  MoveL 9477 to (-30.25, 36.35, 135.08) mm, rotated rx 180 ry 0 rz 180 deg; joints [-35.768, -29.78, 105.46, 71.051, 38.171, -66.408]
  MoveL 9478 to (-30.25, 36.35, 135.08) mm, rotated rx 180 ry 0 rz 180 deg; joints [-35.768, -29.78, 105.46, 71.051, 38.171, -66.408]
  Call Extruder(64.93242)
  MoveL 9479 to (-30.02, 36.28, 135.08) mm, rotated rx -180 ry 0 rz -180 deg; joints [-35.728, -29.761, 105.45, 71.036, 38.13, -66.402]
  MoveL 9480 to (-30.02, 36.28, 135.08) mm, rotated rx -180 ry 0 rz -180 deg; joints [-35.728, -29.761, 105.45, 71.036, 38.13, -66.402]
  Call Extruder(65.06180)
  MoveL 9481 to (-29.8, 36.22, 135.08) mm, rotated rx -180 ry 0 rz 180 deg; joints [-35.688, -29.741, 105.44, 71.022, 38.09, -66.397]
  MoveL 9482 to (-29.8, 36.22, 135.08) mm, rotated rx -180 ry 0 rz 180 deg; joints [-35.688, -29.741, 105.44, 71.022, 38.09, -66.397]
  Call Extruder(65.18377)
  MoveL 9483 to (-29.59, 36.16, 135.08) mm, rotated rx 180 ry 0 rz 180 deg; joints [-35.651, -29.721, 105.43, 71.009, 38.053, -66.393]
  MoveL 9484 to (-29.59, 36.16, 135.08) mm, rotated rx 180 ry 0 rz 180 deg; joints [-35.651, -29.721, 105.43, 71.009, 38.053, -66.393]
  Call Extruder(65.29861)
  MoveL 9485 to (-29.38, 36.12, 135.08) mm, rotated rx -180 ry 0 rz 180 deg; joints [-35.617, -29.701, 105.42, 70.999, 38.019, -66.39]
  MoveL 9486 to (-29.38, 36.12, 135.08) mm, rotated rx -180 ry 0 rz 180 deg; joints [-35.617, -29.701, 105.42, 70.999, 38.019, -66.39]
  Call Extruder(65.41301)
  MoveL 9487 to (-29.18, 36.07, 135.08) mm, rotated rx 180 ry 0 rz 180 deg; joints [-35.584, -29.682, 105.41, 70.989, 37.986, -66.388]
  MoveL 9488 to (-29.18, 36.07, 135.08) mm, rotated rx 180 ry 0 rz 180 deg; joints [-35.584, -29.682, 105.41, 70.989, 37.986, -66.388]
  Call Extruder(65.52695)
  MoveL 9489 to (-28.97, 36.03, 135.08) mm, rotated rx 180 ry 0 rz -180 deg; joints [-35.55, -29.662, 105.4, 70.979, 37.952, -66.385]
  MoveL 9490 to (-28.97, 36.03, 135.08) mm, rotated rx 180 ry 0 rz -180 deg; joints [-35.55, -29.662, 105.4, 70.979, 37.952, -66.385]
  Call Extruder(65.64044)
  MoveL 9491 to (-28.77, 35.98, 135.08) mm, rotated rx -180 ry 0 rz 180 deg; joints [-35.517, -29.642, 105.39, 70.969, 37.918, -66.383]
  MoveL 9492 to (-28.77, 35.98, 135.08) mm, rotated rx -180 ry 0 rz 180 deg; joints [-35.517, -29.642, 105.39, 70.969, 37.918, -66.383]
  Call Extruder(65.77772)
  MoveL 9493 to (-28.52, 35.93, 135.08) mm, rotated rx -180 ry 0 rz 180 deg; joints [-35.477, -29.618, 105.377, 70.957, 37.877, -66.38]
  MoveL 9494 to (-28.52, 35.93, 135.08) mm, rotated rx -180 ry 0 rz 180 deg; joints [-35.477, -29.618, 105.377, 70.957, 37.877, -66.38]
  Call Extruder(65.91440)
  MoveL 9495 to (-28.27, 35.88, 135.08) mm, rotated rx 180 ry 0 rz 180 deg; joints [-35.437, -29.593, 105.365, 70.945, 37.837, -66.378]
  MoveL 9496 to (-28.27, 35.88, 135.08) mm, rotated rx 180 ry 0 rz 180 deg; joints [-35.437, -29.593, 105.365, 70.945, 37.837, -66.378]
  Call Extruder(66.05046)
  MoveL 9497 to (-28.02, 35.83, 135.08) mm, rotated rx 180 ry 0 rz -180 deg; joints [-35.397, -29.569, 105.352, 70.934, 37.796, -66.376]
  MoveL 9498 to (-28.02, 35.83, 135.08) mm, rotated rx 180 ry 0 rz -180 deg; joints [-35.397, -29.569, 105.352, 70.934, 37.796, -66.376]
  Call Extruder(66.18591)
  MoveL 9499 to (-27.77, 35.78, 135.08) mm, rotated rx 180 ry 0 rz 180 deg; joints [-35.357, -29.544, 105.339, 70.922, 37.756, -66.374]
  MoveL 9500 to (-27.77, 35.78, 135.08) mm, rotated rx 180 ry 0 rz 180 deg; joints [-35.357, -29.544, 105.339, 70.922, 37.756, -66.374]
  Call Extruder(66.32075)
  MoveL 9501 to (-27.52, 35.73, 135.08) mm, rotated rx -180 ry 0 rz -180 deg; joints [-35.317, -29.52, 105.327, 70.911, 37.716, -66.371]
  MoveL 9502 to (-27.52, 35.73, 135.08) mm, rotated rx -180 ry 0 rz -180 deg; joints [-35.317, -29.52, 105.327, 70.911, 37.716, -66.371]
  Call Extruder(66.45498)
  MoveL 9503 to (-27.27, 35.68, 135.08) mm, rotated rx 180 ry 0 rz 180 deg; joints [-35.277, -29.496, 105.314, 70.899, 37.675, -66.369]
  MoveL 9504 to (-27.27, 35.68, 135.08) mm, rotated rx 180 ry 0 rz 180 deg; joints [-35.277, -29.496, 105.314, 70.899, 37.675, -66.369]
  Call Extruder(66.58860)
  MoveL 9505 to (-27.03, 35.64, 135.08) mm, rotated rx 180 ry 0 rz 180 deg; joints [-35.238, -29.471, 105.302, 70.888, 37.635, -66.367]
  MoveL 9506 to (-27.03, 35.64, 135.08) mm, rotated rx 180 ry 0 rz 180 deg; joints [-35.238, -29.471, 105.302, 70.888, 37.635, -66.367]
  Call Extruder(66.75070)
  MoveL 9507 to (-26.72, 35.59, 135.08) mm, rotated rx -180 ry 0 rz 180 deg; joints [-35.191, -29.44, 105.286, 70.875, 37.587, -66.366]
  MoveL 9508 to (-26.72, 35.59, 135.08) mm, rotated rx -180 ry 0 rz 180 deg; joints [-35.191, -29.44, 105.286, 70.875, 37.587, -66.366]
  Call Extruder(66.91207)
  MoveL 9509 to (-26.41, 35.54, 135.08) mm, rotated rx -180 ry 0 rz 180 deg; joints [-35.145, -29.409, 105.269, 70.864, 37.54, -66.365]
  MoveL 9510 to (-26.41, 35.54, 135.08) mm, rotated rx -180 ry 0 rz 180 deg; joints [-35.145, -29.409, 105.269, 70.864, 37.54, -66.365]
  Call Extruder(67.07271)
  MoveL 9511 to (-26.11, 35.49, 135.08) mm, rotated rx 180 ry 0 rz 180 deg; joints [-35.098, -29.377, 105.253, 70.852, 37.493, -66.364]
  MoveL 9512 to (-26.11, 35.49, 135.08) mm, rotated rx 180 ry 0 rz 180 deg; joints [-35.098, -29.377, 105.253, 70.852, 37.493, -66.364]
  Call Extruder(67.23263)
  MoveL 9513 to (-25.8, 35.44, 135.08) mm, rotated rx 180 ry 0 rz 180 deg; joints [-35.052, -29.346, 105.237, 70.84, 37.445, -66.364]
  MoveL 9514 to (-25.8, 35.44, 135.08) mm, rotated rx 180 ry 0 rz 180 deg; joints [-35.052, -29.346, 105.237, 70.84, 37.445, -66.364]
  Call Extruder(67.39181)
  MoveL 9515 to (-25.5, 35.39, 135.08) mm, rotated rx -180 ry 0 rz 180 deg; joints [-35.006, -29.315, 105.221, 70.828, 37.398, -66.363]
  MoveL 9516 to (-25.5, 35.39, 135.08) mm, rotated rx -180 ry 0 rz 180 deg; joints [-35.006, -29.315, 105.221, 70.828, 37.398, -66.363]
  Call Extruder(67.55027)
  MoveL 9517 to (-25.19, 35.34, 135.08) mm, rotated rx 180 ry 0 rz 180 deg; joints [-34.96, -29.284, 105.205, 70.816, 37.351, -66.362]
  MoveL 9518 to (-25.19, 35.34, 135.08) mm, rotated rx 180 ry 0 rz 180 deg; joints [-34.96, -29.284, 105.205, 70.816, 37.351, -66.362]
  Call Extruder(67.74915)
  MoveL 9519 to (-24.8, 35.3, 135.08) mm, rotated rx 180 ry 0 rz 180 deg; joints [-34.904, -29.243, 105.184, 70.804, 37.294, -66.364]
  MoveL 9520 to (-24.8, 35.3, 135.08) mm, rotated rx 180 ry 0 rz 180 deg; joints [-34.904, -29.243, 105.184, 70.804, 37.294, -66.364]
  Call Extruder(67.94716)
  MoveL 9521 to (-24.42, 35.25, 135.08) mm, rotated rx -180 ry 0 rz 180 deg; joints [-34.849, -29.202, 105.162, 70.791, 37.236, -66.365]
  MoveL 9522 to (-24.42, 35.25, 135.08) mm, rotated rx -180 ry 0 rz 180 deg; joints [-34.849, -29.202, 105.162, 70.791, 37.236, -66.365]
  Call Extruder(68.14430)
  MoveL 9523 to (-24.03, 35.21, 135.08) mm, rotated rx 180 ry 0 rz 180 deg; joints [-34.794, -29.161, 105.141, 70.779, 37.179, -66.367]
  MoveL 9524 to (-24.03, 35.21, 135.08) mm, rotated rx 180 ry 0 rz 180 deg; joints [-34.794, -29.161, 105.141, 70.779, 37.179, -66.367]
  Call Extruder(68.34057)
  MoveL 9525 to (-23.64, 35.16, 135.08) mm, rotated rx -180 ry 0 rz 180 deg; joints [-34.738, -29.12, 105.119, 70.767, 37.122, -66.368]
  MoveL 9526 to (-23.64, 35.16, 135.08) mm, rotated rx -180 ry 0 rz 180 deg; joints [-34.738, -29.12, 105.119, 70.767, 37.122, -66.368]
  Call Extruder(68.58626)
  MoveL 9527 to (-23.15, 35.11, 135.08) mm, rotated rx -180 ry 0 rz 180 deg; joints [-34.671, -29.067, 105.092, 70.754, 37.052, -66.372]
  MoveL 9528 to (-23.15, 35.11, 135.08) mm, rotated rx -180 ry 0 rz 180 deg; joints [-34.671, -29.067, 105.092, 70.754, 37.052, -66.372]
  Call Extruder(68.88099)
  MoveL 9529 to (-22.56, 35.07, 135.08) mm, rotated rx 180 ry 0 rz 180 deg; joints [-34.592, -29.002, 105.058, 70.739, 36.969, -66.378]
  MoveL 9530 to (-22.56, 35.07, 135.08) mm, rotated rx 180 ry 0 rz 180 deg; joints [-34.592, -29.002, 105.058, 70.739, 36.969, -66.378]
  Call Extruder(69.17439)
  MoveL 9531 to (-21.97, 35.02, 135.08) mm, rotated rx 180 ry 0 rz 180 deg; joints [-34.512, -28.938, 105.024, 70.725, 36.886, -66.384]
  MoveL 9532 to (-21.97, 35.02, 135.08) mm, rotated rx 180 ry 0 rz 180 deg; joints [-34.512, -28.938, 105.024, 70.725, 36.886, -66.384]
  Call Extruder(69.60772)
  MoveL 9533 to (-21.1, 34.97, 135.08) mm, rotated rx 180 ry 0 rz 180 deg; joints [-34.399, -28.84, 104.973, 70.708, 36.767, -66.397]
  MoveL 9534 to (-21.1, 34.97, 135.08) mm, rotated rx 180 ry 0 rz 180 deg; joints [-34.399, -28.84, 104.973, 70.708, 36.767, -66.397]
  Call Extruder(70.17988)
  MoveL 9535 to (-19.94, 34.93, 135.08) mm, rotated rx 180 ry 0 rz 180 deg; joints [-34.253, -28.708, 104.904, 70.689, 36.613, -66.416]
  MoveL 9536 to (-19.94, 34.93, 135.08) mm, rotated rx 180 ry 0 rz 180 deg; joints [-34.253, -28.708, 104.904, 70.689, 36.613, -66.416]
  Call Extruder(70.60771)
  MoveL 9537 to (-19.06, 34.91, 135.08) mm, rotated rx 180 ry 0 rz 180 deg; joints [-34.146, -28.608, 104.85, 70.677, 36.499, -66.434]
  Call Extruder(187.25639)
  MoveL 9538 to (219.06, 34.91, 135.08) mm, rotated rx -180 ry 0 rz 180 deg; joints [-18.248, 3.511, 79.317, 69.262, 19.562, -68.108]
  MoveL 9539 to (219.06, 34.91, 135.08) mm, rotated rx -180 ry 0 rz 180 deg; joints [-18.248, 3.511, 79.317, 69.262, 19.562, -68.108]
  Call Extruder(187.97196)
  MoveL 9540 to (220.52, 34.95, 135.08) mm, rotated rx 180 ry 0 rz 180 deg; joints [-18.199, 3.735, 79.08, 69.172, 19.522, -68.02]
  MoveL 9541 to (220.52, 34.95, 135.08) mm, rotated rx 180 ry 0 rz 180 deg; joints [-18.199, 3.735, 79.08, 69.172, 19.522, -68.02]
  Call Extruder(188.54670)
  MoveL 9542 to (221.68, 35, 135.08) mm, rotated rx 180 ry 0 rz 180 deg; joints [-18.162, 3.916, 78.888, 69.101, 19.491, -67.949]
  MoveL 9543 to (221.68, 35, 135.08) mm, rotated rx 180 ry 0 rz 180 deg; joints [-18.162, 3.916, 78.888, 69.101, 19.491, -67.949]
  Call Extruder(188.84009)
  MoveL 9544 to (222.27, 35.04, 135.08) mm, rotated rx -180 ry 0 rz 180 deg; joints [-18.146, 4.008, 78.789, 69.066, 19.478, -67.915]
  MoveL 9545 to (222.27, 35.04, 135.08) mm, rotated rx -180 ry 0 rz 180 deg; joints [-18.146, 4.008, 78.789, 69.066, 19.478, -67.915]
  Call Extruder(189.13482)
  MoveL 9546 to (222.86, 35.09, 135.08) mm, rotated rx -180 ry 0 rz -180 deg; joints [-18.13, 4.101, 78.691, 69.032, 19.465, -67.88]
  MoveL 9547 to (222.86, 35.09, 135.08) mm, rotated rx -180 ry 0 rz -180 deg; joints [-18.13, 4.101, 78.691, 69.032, 19.465, -67.88]
  Call Extruder(189.43087)
  MoveL 9548 to (223.45, 35.14, 135.08) mm, rotated rx 180 ry 0 rz 180 deg; joints [-18.113, 4.194, 78.591, 68.997, 19.452, -67.846]
  MoveL 9549 to (223.45, 35.14, 135.08) mm, rotated rx 180 ry 0 rz 180 deg; joints [-18.113, 4.194, 78.591, 68.997, 19.452, -67.846]
  Call Extruder(189.62715)
  MoveL 9550 to (223.84, 35.18, 135.08) mm, rotated rx -180 ry 0 rz 180 deg; joints [-18.104, 4.256, 78.525, 68.976, 19.446, -67.824]
  MoveL 9551 to (223.84, 35.18, 135.08) mm, rotated rx -180 ry 0 rz 180 deg; joints [-18.104, 4.256, 78.525, 68.976, 19.446, -67.824]
  Call Extruder(189.82429)
  MoveL 9552 to (224.22, 35.23, 135.08) mm, rotated rx 180 ry 0 rz 180 deg; joints [-18.095, 4.318, 78.459, 68.954, 19.439, -67.802]
  MoveL 9553 to (224.22, 35.23, 135.08) mm, rotated rx 180 ry 0 rz 180 deg; joints [-18.095, 4.318, 78.459, 68.954, 19.439, -67.802]
  Call Extruder(190.02230)
  MoveL 9554 to (224.61, 35.27, 135.08) mm, rotated rx -180 ry 0 rz 180 deg; joints [-18.087, 4.38, 78.393, 68.932, 19.432, -67.78]
  MoveL 9555 to (224.61, 35.27, 135.08) mm, rotated rx -180 ry 0 rz 180 deg; joints [-18.087, 4.38, 78.393, 68.932, 19.432, -67.78]
  Call Extruder(190.22117)
  MoveL 9556 to (225, 35.32, 135.08) mm, rotated rx 180 ry 0 rz -180 deg; joints [-18.078, 4.442, 78.326, 68.91, 19.426, -67.758]
  MoveL 9557 to (225, 35.32, 135.08) mm, rotated rx 180 ry 0 rz -180 deg; joints [-18.078, 4.442, 78.326, 68.91, 19.426, -67.758]
  Call Extruder(190.40025)
  MoveL 9558 to (225.34, 35.37, 135.08) mm, rotated rx 180 ry 0 rz 180 deg; joints [-18.07, 4.497, 78.267, 68.891, 19.42, -67.739]
  MoveL 9559 to (225.34, 35.37, 135.08) mm, rotated rx 180 ry 0 rz 180 deg; joints [-18.07, 4.497, 78.267, 68.891, 19.42, -67.739]
  Call Extruder(190.55944)
  MoveL 9560 to (225.65, 35.42, 135.08) mm, rotated rx 180 ry 0 rz 180 deg; joints [-18.065, 4.547, 78.213, 68.875, 19.417, -67.723]
  MoveL 9561 to (225.65, 35.42, 135.08) mm, rotated rx 180 ry 0 rz 180 deg; joints [-18.065, 4.547, 78.213, 68.875, 19.417, -67.723]
  Call Extruder(190.71935)
  MoveL 9562 to (225.96, 35.47, 135.08) mm, rotated rx 180 ry 0 rz 180 deg; joints [-18.059, 4.597, 78.16, 68.859, 19.413, -67.706]
  MoveL 9563 to (225.96, 35.47, 135.08) mm, rotated rx 180 ry 0 rz 180 deg; joints [-18.059, 4.597, 78.16, 68.859, 19.413, -67.706]
  Call Extruder(190.87999)
  MoveL 9564 to (226.26, 35.51, 135.08) mm, rotated rx 180 ry 0 rz 180 deg; joints [-18.054, 4.646, 78.107, 68.843, 19.409, -67.69]
  MoveL 9565 to (226.26, 35.51, 135.08) mm, rotated rx 180 ry 0 rz 180 deg; joints [-18.054, 4.646, 78.107, 68.843, 19.409, -67.69]
  Call Extruder(191.04136)
  MoveL 9566 to (226.57, 35.56, 135.08) mm, rotated rx 180 ry 0 rz 180 deg; joints [-18.048, 4.696, 78.053, 68.826, 19.405, -67.673]
  MoveL 9567 to (226.57, 35.56, 135.08) mm, rotated rx 180 ry 0 rz 180 deg; joints [-18.048, 4.696, 78.053, 68.826, 19.405, -67.673]
  Call Extruder(191.20345)
  MoveL 9568 to (226.87, 35.61, 135.08) mm, rotated rx -180 ry 0 rz 180 deg; joints [-18.042, 4.745, 78, 68.81, 19.401, -67.657]
  MoveL 9569 to (226.87, 35.61, 135.08) mm, rotated rx -180 ry 0 rz 180 deg; joints [-18.042, 4.745, 78, 68.81, 19.401, -67.657]
  Call Extruder(191.35165)
  MoveL 9570 to (227.15, 35.66, 135.08) mm, rotated rx -180 ry 0 rz 180 deg; joints [-18.038, 4.791, 77.951, 68.795, 19.398, -67.642]
  MoveL 9571 to (227.15, 35.66, 135.08) mm, rotated rx -180 ry 0 rz 180 deg; joints [-18.038, 4.791, 77.951, 68.795, 19.398, -67.642]
  Call Extruder(191.48588)
  MoveL 9572 to (227.4, 35.71, 135.08) mm, rotated rx 180 ry 0 rz 180 deg; joints [-18.034, 4.832, 77.907, 68.783, 19.396, -67.629]
  MoveL 9573 to (227.4, 35.71, 135.08) mm, rotated rx 180 ry 0 rz 180 deg; joints [-18.034, 4.832, 77.907, 68.783, 19.396, -67.629]
  Call Extruder(191.62072)
  MoveL 9574 to (227.65, 35.76, 135.08) mm, rotated rx -180 ry 0 rz 180 deg; joints [-18.031, 4.872, 77.863, 68.77, 19.394, -67.616]
  MoveL 9575 to (227.65, 35.76, 135.08) mm, rotated rx -180 ry 0 rz 180 deg; joints [-18.031, 4.872, 77.863, 68.77, 19.394, -67.616]
  Call Extruder(191.75618)
  MoveL 9576 to (227.9, 35.81, 135.08) mm, rotated rx 180 ry 0 rz 180 deg; joints [-18.027, 4.913, 77.819, 68.758, 19.392, -67.603]
  MoveL 9577 to (227.9, 35.81, 135.08) mm, rotated rx 180 ry 0 rz 180 deg; joints [-18.027, 4.913, 77.819, 68.758, 19.392, -67.603]
  Call Extruder(191.89224)
  MoveL 9578 to (228.15, 35.86, 135.08) mm, rotated rx 180 ry 0 rz -180 deg; joints [-18.024, 4.954, 77.774, 68.745, 19.39, -67.59]
  MoveL 9579 to (228.15, 35.86, 135.08) mm, rotated rx 180 ry 0 rz -180 deg; joints [-18.024, 4.954, 77.774, 68.745, 19.39, -67.59]
  Call Extruder(192.02891)
  MoveL 9580 to (228.4, 35.91, 135.08) mm, rotated rx 180 ry 0 rz -180 deg; joints [-18.02, 4.996, 77.73, 68.732, 19.388, -67.577]
  MoveL 9581 to (228.4, 35.91, 135.08) mm, rotated rx 180 ry 0 rz -180 deg; joints [-18.02, 4.996, 77.73, 68.732, 19.388, -67.577]
  Call Extruder(192.16620)
  MoveL 9582 to (228.64, 35.96, 135.08) mm, rotated rx 180 ry 0 rz 180 deg; joints [-18.017, 5.037, 77.685, 68.719, 19.386, -67.564]
  MoveL 9583 to (228.64, 35.96, 135.08) mm, rotated rx 180 ry 0 rz 180 deg; joints [-18.017, 5.037, 77.685, 68.719, 19.386, -67.564]
  Call Extruder(192.29187)
  MoveL 9584 to (228.87, 36, 135.08) mm, rotated rx 180 ry 0 rz 180 deg; joints [-18.014, 5.074, 77.645, 68.708, 19.385, -67.552]
  MoveL 9585 to (228.87, 36, 135.08) mm, rotated rx 180 ry 0 rz 180 deg; joints [-18.014, 5.074, 77.645, 68.708, 19.385, -67.552]
  Call Extruder(192.40582)
  MoveL 9586 to (229.08, 36.05, 135.08) mm, rotated rx -180 ry 0 rz 180 deg; joints [-18.012, 5.108, 77.608, 68.698, 19.383, -67.542]
  MoveL 9587 to (229.08, 36.05, 135.08) mm, rotated rx -180 ry 0 rz 180 deg; joints [-18.012, 5.108, 77.608, 68.698, 19.383, -67.542]
  Call Extruder(192.52022)
  MoveL 9588 to (229.28, 36.09, 135.08) mm, rotated rx 180 ry 0 rz 180 deg; joints [-18.009, 5.142, 77.572, 68.687, 19.382, -67.531]
  MoveL 9589 to (229.28, 36.09, 135.08) mm, rotated rx 180 ry 0 rz 180 deg; joints [-18.009, 5.142, 77.572, 68.687, 19.382, -67.531]
  Call Extruder(192.63507)
  MoveL 9590 to (229.48, 36.14, 135.08) mm, rotated rx 180 ry 0 rz 180 deg; joints [-18.007, 5.176, 77.535, 68.677, 19.381, -67.521]
  MoveL 9591 to (229.48, 36.14, 135.08) mm, rotated rx 180 ry 0 rz 180 deg; joints [-18.007, 5.176, 77.535, 68.677, 19.381, -67.521]
  Call Extruder(192.75038)
  MoveL 9592 to (229.69, 36.18, 135.08) mm, rotated rx 180 ry 0 rz 180 deg; joints [-18.005, 5.21, 77.498, 68.667, 19.38, -67.51]
  MoveL 9593 to (229.69, 36.18, 135.08) mm, rotated rx 180 ry 0 rz 180 deg; joints [-18.005, 5.21, 77.498, 68.667, 19.38, -67.51]
  Call Extruder(192.82364)
  MoveL 9594 to (229.81, 36.22, 135.08) mm, rotated rx -180 ry 0 rz 180 deg; joints [-18.004, 5.231, 77.475, 68.661, 19.38, -67.504]
  MoveL 9595 to (229.81, 36.22, 135.08) mm, rotated rx -180 ry 0 rz 180 deg; joints [-18.004, 5.231, 77.475, 68.661, 19.38, -67.504]
  Call Extruder(192.95114)
  MoveL 9596 to (230.04, 36.29, 135.08) mm, rotated rx 180 ry 0 rz 180 deg; joints [-18.004, 5.269, 77.434, 68.652, 19.381, -67.495]
  MoveL 9597 to (230.04, 36.29, 135.08) mm, rotated rx 180 ry 0 rz 180 deg; joints [-18.004, 5.269, 77.434, 68.652, 19.381, -67.495]
  Call Extruder(193.07920)
  MoveL 9598 to (230.26, 36.35, 135.08) mm, rotated rx 180 ry 0 rz 180 deg; joints [-18.003, 5.306, 77.393, 68.643, 19.382, -67.485]
  MoveL 9599 to (230.26, 36.35, 135.08) mm, rotated rx 180 ry 0 rz 180 deg; joints [-18.003, 5.306, 77.393, 68.643, 19.382, -67.485]
  Call Extruder(193.20780)
  MoveL 9600 to (230.48, 36.42, 135.08) mm, rotated rx -180 ry 0 rz 180 deg; joints [-18.003, 5.344, 77.353, 68.634, 19.382, -67.475]
  MoveL 9601 to (230.48, 36.42, 135.08) mm, rotated rx -180 ry 0 rz 180 deg; joints [-18.003, 5.344, 77.353, 68.634, 19.382, -67.475]
  Call Extruder(193.33694)
  MoveL 9602 to (230.69, 36.49, 135.08) mm, rotated rx 180 ry 0 rz 180 deg; joints [-18.002, 5.381, 77.312, 68.625, 19.383, -67.466]
  MoveL 9603 to (230.69, 36.49, 135.08) mm, rotated rx 180 ry 0 rz 180 deg; joints [-18.002, 5.381, 77.312, 68.625, 19.383, -67.466]
  Call Extruder(193.44884)
  MoveL 9604 to (230.88, 36.55, 135.08) mm, rotated rx 180 ry 0 rz 180 deg; joints [-18.002, 5.413, 77.277, 68.617, 19.384, -67.458]
  MoveL 9605 to (230.88, 36.55, 135.08) mm, rotated rx 180 ry 0 rz 180 deg; joints [-18.002, 5.413, 77.277, 68.617, 19.384, -67.458]
  Call Extruder(193.56118)
  MoveL 9606 to (231.07, 36.61, 135.08) mm, rotated rx -180 ry 0 rz -180 deg; joints [-18.002, 5.446, 77.241, 68.609, 19.385, -67.45]
  MoveL 9607 to (231.07, 36.61, 135.08) mm, rotated rx -180 ry 0 rz -180 deg; joints [-18.002, 5.446, 77.241, 68.609, 19.385, -67.45]
  Call Extruder(193.67397)
  MoveL 9608 to (231.26, 36.67, 135.08) mm, rotated rx -180 ry 0 rz 180 deg; joints [-18.002, 5.478, 77.206, 68.602, 19.386, -67.442]
  MoveL 9609 to (231.26, 36.67, 135.08) mm, rotated rx -180 ry 0 rz 180 deg; joints [-18.002, 5.478, 77.206, 68.602, 19.386, -67.442]
  Call Extruder(193.78720)
  MoveL 9610 to (231.45, 36.73, 135.08) mm, rotated rx 180 ry 0 rz 180 deg; joints [-18.002, 5.511, 77.171, 68.594, 19.387, -67.433]
  MoveL 9611 to (231.45, 36.73, 135.08) mm, rotated rx 180 ry 0 rz 180 deg; joints [-18.002, 5.511, 77.171, 68.594, 19.387, -67.433]
  Call Extruder(193.90088)
  MoveL 9612 to (231.64, 36.79, 135.08) mm, rotated rx 180 ry 0 rz 180 deg; joints [-18.002, 5.543, 77.136, 68.587, 19.388, -67.425]
  MoveL 9613 to (231.64, 36.79, 135.08) mm, rotated rx 180 ry 0 rz 180 deg; joints [-18.002, 5.543, 77.136, 68.587, 19.388, -67.425]
  Call Extruder(194.08284)
  MoveL 9614 to (231.93, 36.91, 135.08) mm, rotated rx 180 ry 0 rz 180 deg; joints [-18.005, 5.594, 77.079, 68.577, 19.393, -67.415]
  MoveL 9615 to (231.93, 36.91, 135.08) mm, rotated rx 180 ry 0 rz 180 deg; joints [-18.005, 5.594, 77.079, 68.577, 19.393, -67.415]
  Call Extruder(194.26556)
  MoveL 9616 to (232.22, 37.04, 135.08) mm, rotated rx 180 ry 0 rz 180 deg; joints [-18.008, 5.646, 77.023, 68.568, 19.397, -67.405]
  MoveL 9617 to (232.22, 37.04, 135.08) mm, rotated rx 180 ry 0 rz 180 deg; joints [-18.008, 5.646, 77.023, 68.568, 19.397, -67.405]
  Call Extruder(194.43598)
  MoveL 9618 to (232.49, 37.15, 135.08) mm, rotated rx -180 ry 0 rz 180 deg; joints [-18.011, 5.694, 76.971, 68.56, 19.401, -67.396]
  MoveL 9619 to (232.49, 37.15, 135.08) mm, rotated rx -180 ry 0 rz 180 deg; joints [-18.011, 5.694, 76.971, 68.56, 19.401, -67.396]
  Call Extruder(194.59398)
  MoveL 9620 to (232.74, 37.26, 135.08) mm, rotated rx 180 ry 0 rz -180 deg; joints [-18.013, 5.738, 76.923, 68.552, 19.405, -67.387]
  MoveL 9621 to (232.74, 37.26, 135.08) mm, rotated rx 180 ry 0 rz -180 deg; joints [-18.013, 5.738, 76.923, 68.552, 19.405, -67.387]
  Call Extruder(194.75258)
  MoveL 9622 to (232.99, 37.36, 135.08) mm, rotated rx -180 ry 0 rz 180 deg; joints [-18.016, 5.782, 76.874, 68.545, 19.409, -67.379]
  MoveL 9623 to (232.99, 37.36, 135.08) mm, rotated rx -180 ry 0 rz 180 deg; joints [-18.016, 5.782, 76.874, 68.545, 19.409, -67.379]
  Call Extruder(194.95874)
  MoveL 9624 to (233.29, 37.54, 135.08) mm, rotated rx 180 ry 0 rz 180 deg; joints [-18.024, 5.838, 76.813, 68.54, 19.419, -67.373]
  MoveL 9625 to (233.29, 37.54, 135.08) mm, rotated rx 180 ry 0 rz 180 deg; joints [-18.024, 5.838, 76.813, 68.54, 19.419, -67.373]
  Call Extruder(195.16569)
  MoveL 9626 to (233.6, 37.71, 135.08) mm, rotated rx 180 ry 0 rz 180 deg; joints [-18.033, 5.895, 76.751, 68.535, 19.429, -67.367]
  MoveL 9627 to (233.6, 37.71, 135.08) mm, rotated rx 180 ry 0 rz 180 deg; joints [-18.033, 5.895, 76.751, 68.535, 19.429, -67.367]
  Call Extruder(195.37341)
  MoveL 9628 to (233.9, 37.89, 135.08) mm, rotated rx 180 ry 0 rz 180 deg; joints [-18.041, 5.951, 76.689, 68.531, 19.438, -67.361]
  MoveL 9629 to (233.9, 37.89, 135.08) mm, rotated rx 180 ry 0 rz 180 deg; joints [-18.041, 5.951, 76.689, 68.531, 19.438, -67.361]
  Call Extruder(195.58192)
  MoveL 9630 to (234.21, 38.07, 135.08) mm, rotated rx 180 ry 0 rz -180 deg; joints [-18.049, 6.007, 76.627, 68.526, 19.448, -67.354]
  MoveL 9631 to (234.21, 38.07, 135.08) mm, rotated rx 180 ry 0 rz -180 deg; joints [-18.049, 6.007, 76.627, 68.526, 19.448, -67.354]
  Call Extruder(195.76146)
  MoveL 9632 to (234.45, 38.24, 135.08) mm, rotated rx 180 ry 0 rz 180 deg; joints [-18.06, 6.055, 76.575, 68.526, 19.459, -67.353]
  MoveL 9633 to (234.45, 38.24, 135.08) mm, rotated rx 180 ry 0 rz 180 deg; joints [-18.06, 6.055, 76.575, 68.526, 19.459, -67.353]
  Call Extruder(196.09487)
  MoveL 9634 to (234.9, 38.57, 135.08) mm, rotated rx 180 ry 0 rz 180 deg; joints [-18.079, 6.142, 76.48, 68.525, 19.48, -67.35]
  MoveL 9635 to (234.9, 38.57, 135.08) mm, rotated rx 180 ry 0 rz 180 deg; joints [-18.079, 6.142, 76.48, 68.525, 19.48, -67.35]
  Call Extruder(196.42947)
  MoveL 9636 to (235.35, 38.9, 135.08) mm, rotated rx 180 ry 0 rz -180 deg; joints [-18.099, 6.229, 76.384, 68.525, 19.502, -67.347]
  Call Extruder(197.25742)
  MoveL 9637 to (236.39, 39.81, 135.08) mm, rotated rx 180 ry 0 rz 180 deg; joints [-18.16, 6.438, 76.153, 68.539, 19.566, -67.354]
  Call Extruder(198.08537)
  MoveL 9638 to (237.3, 40.85, 135.08) mm, rotated rx 180 ry 0 rz -180 deg; joints [-18.24, 6.634, 75.936, 68.575, 19.647, -67.381]
  Call Extruder(198.25267)
  MoveL 9639 to (237.47, 41.07, 135.08) mm, rotated rx 180 ry 0 rz 180 deg; joints [-18.258, 6.672, 75.895, 68.586, 19.666, -67.39]
  MoveL 9640 to (237.47, 41.07, 135.08) mm, rotated rx 180 ry 0 rz 180 deg; joints [-18.258, 6.672, 75.895, 68.586, 19.666, -67.39]
  Call Extruder(198.58609)
  MoveL 9641 to (237.79, 41.52, 135.08) mm, rotated rx 180 ry 0 rz 180 deg; joints [-18.295, 6.746, 75.812, 68.607, 19.703, -67.407]
  MoveL 9642 to (237.79, 41.52, 135.08) mm, rotated rx 180 ry 0 rz 180 deg; joints [-18.295, 6.746, 75.812, 68.607, 19.703, -67.407]
  Call Extruder(198.91833)
  MoveL 9643 to (238.12, 41.98, 135.08) mm, rotated rx 180 ry 0 rz 180 deg; joints [-18.332, 6.821, 75.728, 68.627, 19.739, -67.423]
  MoveL 9644 to (238.12, 41.98, 135.08) mm, rotated rx 180 ry 0 rz 180 deg; joints [-18.332, 6.821, 75.728, 68.627, 19.739, -67.423]
  Call Extruder(199.03601)
  MoveL 9645 to (238.22, 42.15, 135.08) mm, rotated rx 180 ry 0 rz 180 deg; joints [-18.346, 6.846, 75.701, 68.637, 19.754, -67.431]
  MoveL 9646 to (238.22, 42.15, 135.08) mm, rotated rx 180 ry 0 rz 180 deg; joints [-18.346, 6.846, 75.701, 68.637, 19.754, -67.431]
  Call Extruder(199.24373)
  MoveL 9647 to (238.4, 42.45, 135.08) mm, rotated rx 180 ry 0 rz -180 deg; joints [-18.373, 6.889, 75.653, 68.654, 19.78, -67.446]
  MoveL 9648 to (238.4, 42.45, 135.08) mm, rotated rx 180 ry 0 rz -180 deg; joints [-18.373, 6.889, 75.653, 68.654, 19.78, -67.446]
  Call Extruder(199.45067)
  MoveL 9649 to (238.57, 42.75, 135.08) mm, rotated rx 180 ry 0 rz 180 deg; joints [-18.399, 6.933, 75.605, 68.671, 19.806, -67.461]
  MoveL 9650 to (238.57, 42.75, 135.08) mm, rotated rx 180 ry 0 rz 180 deg; joints [-18.399, 6.933, 75.605, 68.671, 19.806, -67.461]
  Call Extruder(199.65683)
  MoveL 9651 to (238.75, 43.06, 135.08) mm, rotated rx 180 ry 0 rz 180 deg; joints [-18.425, 6.976, 75.556, 68.688, 19.832, -67.475]
  MoveL 9652 to (238.75, 43.06, 135.08) mm, rotated rx 180 ry 0 rz 180 deg; joints [-18.425, 6.976, 75.556, 68.688, 19.832, -67.475]
  Call Extruder(199.83852)
  MoveL 9653 to (238.89, 43.34, 135.08) mm, rotated rx -180 ry 0 rz 180 deg; joints [-18.45, 7.013, 75.515, 68.705, 19.856, -67.489]
  MoveL 9654 to (238.89, 43.34, 135.08) mm, rotated rx -180 ry 0 rz 180 deg; joints [-18.45, 7.013, 75.515, 68.705, 19.856, -67.489]
  Call Extruder(199.99654)
  MoveL 9655 to (239, 43.58, 135.08) mm, rotated rx 180 ry 0 rz 180 deg; joints [-18.472, 7.043, 75.482, 68.721, 19.879, -67.504]
  MoveL 9656 to (239, 43.58, 135.08) mm, rotated rx 180 ry 0 rz 180 deg; joints [-18.472, 7.043, 75.482, 68.721, 19.879, -67.504]
  Call Extruder(200.15395)
  MoveL 9657 to (239.11, 43.83, 135.08) mm, rotated rx 180 ry 0 rz -180 deg; joints [-18.495, 7.073, 75.449, 68.738, 19.901, -67.519]
  MoveL 9658 to (239.11, 43.83, 135.08) mm, rotated rx 180 ry 0 rz -180 deg; joints [-18.495, 7.073, 75.449, 68.738, 19.901, -67.519]
  Call Extruder(200.33666)
  MoveL 9659 to (239.23, 44.13, 135.08) mm, rotated rx -180 ry 0 rz 180 deg; joints [-18.522, 7.107, 75.41, 68.758, 19.927, -67.536]
  MoveL 9660 to (239.23, 44.13, 135.08) mm, rotated rx -180 ry 0 rz 180 deg; joints [-18.522, 7.107, 75.41, 68.758, 19.927, -67.536]
  Call Extruder(200.51862)
  MoveL 9661 to (239.35, 44.42, 135.08) mm, rotated rx 180 ry 0 rz 180 deg; joints [-18.549, 7.141, 75.372, 68.778, 19.953, -67.554]
  MoveL 9662 to (239.35, 44.42, 135.08) mm, rotated rx 180 ry 0 rz 180 deg; joints [-18.549, 7.141, 75.372, 68.778, 19.953, -67.554]
  Call Extruder(200.66595)
  MoveL 9663 to (239.44, 44.66, 135.08) mm, rotated rx 180 ry 0 rz 180 deg; joints [-18.571, 7.168, 75.342, 68.795, 19.975, -67.568]
  MoveL 9664 to (239.44, 44.66, 135.08) mm, rotated rx 180 ry 0 rz 180 deg; joints [-18.571, 7.168, 75.342, 68.795, 19.975, -67.568]
  Call Extruder(200.77919)
  MoveL 9665 to (239.5, 44.85, 135.08) mm, rotated rx -180 ry 0 rz -180 deg; joints [-18.589, 7.188, 75.32, 68.809, 19.992, -67.581]
  MoveL 9666 to (239.5, 44.85, 135.08) mm, rotated rx -180 ry 0 rz -180 deg; joints [-18.589, 7.188, 75.32, 68.809, 19.992, -67.581]
  Call Extruder(200.89198)
  MoveL 9667 to (239.56, 45.03, 135.08) mm, rotated rx 180 ry 0 rz 180 deg; joints [-18.607, 7.207, 75.298, 68.823, 20.01, -67.593]
  MoveL 9668 to (239.56, 45.03, 135.08) mm, rotated rx 180 ry 0 rz 180 deg; joints [-18.607, 7.207, 75.298, 68.823, 20.01, -67.593]
  Call Extruder(201.00432)
  MoveL 9669 to (239.62, 45.22, 135.08) mm, rotated rx 180 ry 0 rz 180 deg; joints [-18.625, 7.227, 75.276, 68.837, 20.027, -67.606]
  MoveL 9670 to (239.62, 45.22, 135.08) mm, rotated rx 180 ry 0 rz 180 deg; joints [-18.625, 7.227, 75.276, 68.837, 20.027, -67.606]
  Call Extruder(201.11622)
  MoveL 9671 to (239.68, 45.41, 135.08) mm, rotated rx 180 ry 0 rz 180 deg; joints [-18.642, 7.246, 75.254, 68.851, 20.044, -67.618]
  MoveL 9672 to (239.68, 45.41, 135.08) mm, rotated rx 180 ry 0 rz 180 deg; joints [-18.642, 7.246, 75.254, 68.851, 20.044, -67.618]
  Call Extruder(201.23762)
  MoveL 9673 to (239.75, 45.62, 135.08) mm, rotated rx 180 ry 0 rz 180 deg; joints [-18.662, 7.268, 75.231, 68.866, 20.063, -67.632]
  MoveL 9674 to (239.75, 45.62, 135.08) mm, rotated rx 180 ry 0 rz 180 deg; joints [-18.662, 7.268, 75.231, 68.866, 20.063, -67.632]
  Call Extruder(201.36842)
  MoveL 9675 to (239.82, 45.84, 135.08) mm, rotated rx 180 ry 0 rz 180 deg; joints [-18.683, 7.29, 75.205, 68.883, 20.084, -67.647]
  MoveL 9676 to (239.82, 45.84, 135.08) mm, rotated rx 180 ry 0 rz 180 deg; joints [-18.683, 7.29, 75.205, 68.883, 20.084, -67.647]
  Call Extruder(201.49864)
  MoveL 9677 to (239.88, 46.06, 135.08) mm, rotated rx 180 ry 0 rz 180 deg; joints [-18.705, 7.313, 75.18, 68.9, 20.105, -67.661]
  MoveL 9678 to (239.88, 46.06, 135.08) mm, rotated rx 180 ry 0 rz 180 deg; joints [-18.705, 7.313, 75.18, 68.9, 20.105, -67.661]
  Call Extruder(201.62830)
  MoveL 9679 to (239.95, 46.29, 135.08) mm, rotated rx 180 ry 0 rz 180 deg; joints [-18.726, 7.335, 75.155, 68.916, 20.125, -67.676]
  MoveL 9680 to (239.95, 46.29, 135.08) mm, rotated rx 180 ry 0 rz 180 deg; joints [-18.726, 7.335, 75.155, 68.916, 20.125, -67.676]
  Call Extruder(201.75740)
  MoveL 9681 to (240.02, 46.51, 135.08) mm, rotated rx 180 ry 0 rz 180 deg; joints [-18.747, 7.358, 75.13, 68.933, 20.146, -67.691]
  MoveL 9682 to (240.02, 46.51, 135.08) mm, rotated rx 180 ry 0 rz 180 deg; joints [-18.747, 7.358, 75.13, 68.933, 20.146, -67.691]
  Call Extruder(201.87246)
  MoveL 9683 to (240.06, 46.72, 135.08) mm, rotated rx -180 ry 0 rz 180 deg; joints [-18.767, 7.376, 75.11, 68.949, 20.165, -67.706]
  MoveL 9684 to (240.06, 46.72, 135.08) mm, rotated rx -180 ry 0 rz 180 deg; joints [-18.767, 7.376, 75.11, 68.949, 20.165, -67.706]
  Call Extruder(201.98706)
  MoveL 9685 to (240.11, 46.92, 135.08) mm, rotated rx 180 ry 0 rz 180 deg; joints [-18.787, 7.394, 75.09, 68.966, 20.185, -67.721]
  MoveL 9686 to (240.11, 46.92, 135.08) mm, rotated rx 180 ry 0 rz 180 deg; joints [-18.787, 7.394, 75.09, 68.966, 20.185, -67.721]
  Call Extruder(202.10121)
  MoveL 9687 to (240.15, 47.12, 135.08) mm, rotated rx 180 ry 0 rz 180 deg; joints [-18.807, 7.412, 75.07, 68.982, 20.204, -67.735]
  MoveL 9688 to (240.15, 47.12, 135.08) mm, rotated rx 180 ry 0 rz 180 deg; joints [-18.807, 7.412, 75.07, 68.982, 20.204, -67.735]
  Call Extruder(202.21491)
  MoveL 9689 to (240.2, 47.33, 135.08) mm, rotated rx 180 ry 0 rz 180 deg; joints [-18.827, 7.43, 75.049, 68.999, 20.223, -67.75]
  MoveL 9690 to (240.2, 47.33, 135.08) mm, rotated rx 180 ry 0 rz 180 deg; joints [-18.827, 7.43, 75.049, 68.999, 20.223, -67.75]
  Call Extruder(202.34032)
  MoveL 9691 to (240.24, 47.55, 135.08) mm, rotated rx 180 ry 0 rz 180 deg; joints [-18.85, 7.449, 75.027, 69.017, 20.245, -67.767]
  MoveL 9692 to (240.24, 47.55, 135.08) mm, rotated rx 180 ry 0 rz 180 deg; joints [-18.85, 7.449, 75.027, 69.017, 20.245, -67.767]
  Call Extruder(202.47730)
  MoveL 9693 to (240.29, 47.8, 135.08) mm, rotated rx 180 ry 0 rz 180 deg; joints [-18.874, 7.47, 75.004, 69.038, 20.269, -67.785]
  MoveL 9694 to (240.29, 47.8, 135.08) mm, rotated rx 180 ry 0 rz 180 deg; joints [-18.874, 7.47, 75.004, 69.038, 20.269, -67.785]
  Call Extruder(202.61366)
  MoveL 9695 to (240.34, 48.05, 135.08) mm, rotated rx 180 ry 0 rz 180 deg; joints [-18.899, 7.492, 74.98, 69.058, 20.292, -67.803]
  MoveL 9696 to (240.34, 48.05, 135.08) mm, rotated rx 180 ry 0 rz 180 deg; joints [-18.899, 7.492, 74.98, 69.058, 20.292, -67.803]
  Call Extruder(202.74942)
  MoveL 9697 to (240.39, 48.3, 135.08) mm, rotated rx -180 ry 0 rz 180 deg; joints [-18.923, 7.513, 74.956, 69.078, 20.316, -67.821]
  MoveL 9698 to (240.39, 48.3, 135.08) mm, rotated rx -180 ry 0 rz 180 deg; joints [-18.923, 7.513, 74.956, 69.078, 20.316, -67.821]
  Call Extruder(202.88457)
  MoveL 9699 to (240.44, 48.55, 135.08) mm, rotated rx 180 ry 0 rz 180 deg; joints [-18.948, 7.534, 74.932, 69.098, 20.34, -67.839]
  MoveL 9700 to (240.44, 48.55, 135.08) mm, rotated rx 180 ry 0 rz 180 deg; joints [-18.948, 7.534, 74.932, 69.098, 20.34, -67.839]
  Call Extruder(203.01910)
  MoveL 9701 to (240.49, 48.8, 135.08) mm, rotated rx 180 ry 0 rz 180 deg; joints [-18.973, 7.555, 74.908, 69.118, 20.363, -67.857]
  MoveL 9702 to (240.49, 48.8, 135.08) mm, rotated rx 180 ry 0 rz 180 deg; joints [-18.973, 7.555, 74.908, 69.118, 20.363, -67.857]
  Call Extruder(203.15303)
  MoveL 9703 to (240.54, 49.05, 135.08) mm, rotated rx 180 ry 0 rz 180 deg; joints [-18.997, 7.577, 74.884, 69.138, 20.387, -67.875]
  MoveL 9704 to (240.54, 49.05, 135.08) mm, rotated rx 180 ry 0 rz 180 deg; joints [-18.997, 7.577, 74.884, 69.138, 20.387, -67.875]
  Call Extruder(203.30090)
  MoveL 9705 to (240.59, 49.33, 135.08) mm, rotated rx 180 ry 0 rz 180 deg; joints [-19.025, 7.599, 74.859, 69.161, 20.413, -67.895]
  MoveL 9706 to (240.59, 49.33, 135.08) mm, rotated rx 180 ry 0 rz 180 deg; joints [-19.025, 7.599, 74.859, 69.161, 20.413, -67.895]
  Call Extruder(203.46264)
  MoveL 9707 to (240.64, 49.63, 135.08) mm, rotated rx 180 ry 0 rz 180 deg; joints [-19.055, 7.624, 74.832, 69.186, 20.443, -67.918]
  MoveL 9708 to (240.64, 49.63, 135.08) mm, rotated rx 180 ry 0 rz 180 deg; joints [-19.055, 7.624, 74.832, 69.186, 20.443, -67.918]
  Call Extruder(203.62365)
  MoveL 9709 to (240.69, 49.94, 135.08) mm, rotated rx -180 ry 0 rz 180 deg; joints [-19.086, 7.648, 74.804, 69.211, 20.472, -67.941]
  MoveL 9710 to (240.69, 49.94, 135.08) mm, rotated rx -180 ry 0 rz 180 deg; joints [-19.086, 7.648, 74.804, 69.211, 20.472, -67.941]
  Call Extruder(203.78394)
  MoveL 9711 to (240.74, 50.24, 135.08) mm, rotated rx -180 ry 0 rz 180 deg; joints [-19.116, 7.672, 74.777, 69.236, 20.501, -67.963]
  MoveL 9712 to (240.74, 50.24, 135.08) mm, rotated rx -180 ry 0 rz 180 deg; joints [-19.116, 7.672, 74.777, 69.236, 20.501, -67.963]
  Call Extruder(203.94350)
  MoveL 9713 to (240.78, 50.55, 135.08) mm, rotated rx 180 ry 0 rz 180 deg; joints [-19.146, 7.696, 74.75, 69.261, 20.531, -67.986]
  MoveL 9714 to (240.78, 50.55, 135.08) mm, rotated rx 180 ry 0 rz 180 deg; joints [-19.146, 7.696, 74.75, 69.261, 20.531, -67.986]
  Call Extruder(204.10233)
  MoveL 9715 to (240.83, 50.86, 135.08) mm, rotated rx 180 ry 0 rz 180 deg; joints [-19.177, 7.721, 74.722, 69.286, 20.56, -68.008]
  MoveL 9716 to (240.83, 50.86, 135.08) mm, rotated rx 180 ry 0 rz 180 deg; joints [-19.177, 7.721, 74.722, 69.286, 20.56, -68.008]
  Call Extruder(204.28100)
  MoveL 9717 to (240.88, 51.2, 135.08) mm, rotated rx -180 ry 0 rz 180 deg; joints [-19.212, 7.747, 74.692, 69.315, 20.593, -68.034]
  MoveL 9718 to (240.88, 51.2, 135.08) mm, rotated rx -180 ry 0 rz 180 deg; joints [-19.212, 7.747, 74.692, 69.315, 20.593, -68.034]
  Call Extruder(204.47945)
  MoveL 9719 to (240.92, 51.59, 135.08) mm, rotated rx 180 ry 0 rz 180 deg; joints [-19.251, 7.776, 74.66, 69.348, 20.631, -68.063]
  MoveL 9720 to (240.92, 51.59, 135.08) mm, rotated rx 180 ry 0 rz 180 deg; joints [-19.251, 7.776, 74.66, 69.348, 20.631, -68.063]
  Call Extruder(204.67702)
  MoveL 9721 to (240.97, 51.98, 135.08) mm, rotated rx 180 ry 0 rz 180 deg; joints [-19.29, 7.804, 74.628, 69.38, 20.668, -68.092]
  MoveL 9722 to (240.97, 51.98, 135.08) mm, rotated rx 180 ry 0 rz 180 deg; joints [-19.29, 7.804, 74.628, 69.38, 20.668, -68.092]
  Call Extruder(204.87373)
  MoveL 9723 to (241.02, 52.37, 135.08) mm, rotated rx 180 ry 0 rz 180 deg; joints [-19.329, 7.833, 74.596, 69.412, 20.706, -68.121]
  MoveL 9724 to (241.02, 52.37, 135.08) mm, rotated rx 180 ry 0 rz 180 deg; joints [-19.329, 7.833, 74.596, 69.412, 20.706, -68.121]
  Call Extruder(205.06957)
  MoveL 9725 to (241.06, 52.75, 135.08) mm, rotated rx -180 ry 0 rz 180 deg; joints [-19.368, 7.861, 74.564, 69.444, 20.743, -68.15]
  MoveL 9726 to (241.06, 52.75, 135.08) mm, rotated rx -180 ry 0 rz 180 deg; joints [-19.368, 7.861, 74.564, 69.444, 20.743, -68.15]
  Call Extruder(205.36500)
  MoveL 9727 to (241.11, 53.34, 135.08) mm, rotated rx 180 ry 0 rz 180 deg; joints [-19.428, 7.902, 74.518, 69.494, 20.801, -68.195]
  MoveL 9728 to (241.11, 53.34, 135.08) mm, rotated rx 180 ry 0 rz 180 deg; joints [-19.428, 7.902, 74.518, 69.494, 20.801, -68.195]
  Call Extruder(205.65911)
  MoveL 9729 to (241.15, 53.93, 135.08) mm, rotated rx 180 ry 0 rz 180 deg; joints [-19.488, 7.942, 74.473, 69.544, 20.859, -68.24]
  MoveL 9730 to (241.15, 53.93, 135.08) mm, rotated rx 180 ry 0 rz 180 deg; joints [-19.488, 7.942, 74.473, 69.544, 20.859, -68.24]
  Call Extruder(205.95189)
  MoveL 9731 to (241.2, 54.52, 135.08) mm, rotated rx -180 ry 0 rz 180 deg; joints [-19.548, 7.982, 74.428, 69.594, 20.916, -68.285]
  MoveL 9732 to (241.2, 54.52, 135.08) mm, rotated rx -180 ry 0 rz 180 deg; joints [-19.548, 7.982, 74.428, 69.594, 20.916, -68.285]
  Call Extruder(206.52534)
  MoveL 9733 to (241.25, 55.68, 135.08) mm, rotated rx 180 ry 0 rz 180 deg; joints [-19.668, 8.054, 74.346, 69.695, 21.031, -68.375]
  MoveL 9734 to (241.25, 55.68, 135.08) mm, rotated rx 180 ry 0 rz 180 deg; joints [-19.668, 8.054, 74.346, 69.695, 21.031, -68.375]
  Call Extruder(207.23917)
  MoveL 9735 to (241.29, 57.14, 135.08) mm, rotated rx -180 ry 0 rz 180 deg; joints [-19.819, 8.143, 74.246, 69.82, 21.175, -68.488]
  Call Extruder(249.30405)
  MoveL 9736 to (241.29, 142.86, 135.08) mm, rotated rx 180 ry 0 rz 180 deg; joints [-28.232, 14.196, 67.09, 74.243, 29.44, -72.047]
  Call Extruder(249.73248)
  MoveL 9737 to (241.27, 143.74, 135.08) mm, rotated rx 180 ry 0 rz 180 deg; joints [-28.313, 14.268, 67.002, 74.265, 29.521, -72.059]
  MoveL 9738 to (241.27, 143.74, 135.08) mm, rotated rx 180 ry 0 rz 180 deg; joints [-28.313, 14.268, 67.002, 74.265, 29.521, -72.059]
  Call Extruder(250.30594)
  MoveL 9739 to (241.23, 144.9, 135.08) mm, rotated rx 180 ry 0 rz -180 deg; joints [-28.421, 14.36, 66.888, 74.296, 29.631, -72.076]
  MoveL 9740 to (241.23, 144.9, 135.08) mm, rotated rx 180 ry 0 rz -180 deg; joints [-28.421, 14.36, 66.888, 74.296, 29.631, -72.076]
  Call Extruder(250.74027)
  MoveL 9741 to (241.18, 145.77, 135.08) mm, rotated rx 180 ry 0 rz 180 deg; joints [-28.503, 14.428, 66.804, 74.32, 29.713, -72.089]
  MoveL 9742 to (241.18, 145.77, 135.08) mm, rotated rx 180 ry 0 rz 180 deg; joints [-28.503, 14.428, 66.804, 74.32, 29.713, -72.089]
  Call Extruder(251.03438)
  MoveL 9743 to (241.13, 146.36, 135.08) mm, rotated rx -180 ry 0 rz -180 deg; joints [-28.559, 14.471, 66.75, 74.338, 29.769, -72.099]
  MoveL 9744 to (241.13, 146.36, 135.08) mm, rotated rx -180 ry 0 rz -180 deg; joints [-28.559, 14.471, 66.75, 74.338, 29.769, -72.099]
  Call Extruder(251.32982)
  MoveL 9745 to (241.09, 146.95, 135.08) mm, rotated rx 180 ry 0 rz 180 deg; joints [-28.615, 14.515, 66.697, 74.355, 29.825, -72.109]
  MoveL 9746 to (241.09, 146.95, 135.08) mm, rotated rx 180 ry 0 rz 180 deg; joints [-28.615, 14.515, 66.697, 74.355, 29.825, -72.109]
  Call Extruder(251.57607)
  MoveL 9747 to (241.04, 147.44, 135.08) mm, rotated rx 180 ry 0 rz 180 deg; joints [-28.662, 14.55, 66.653, 74.37, 29.872, -72.118]
  MoveL 9748 to (241.04, 147.44, 135.08) mm, rotated rx 180 ry 0 rz 180 deg; joints [-28.662, 14.55, 66.653, 74.37, 29.872, -72.118]
  Call Extruder(251.77278)
  MoveL 9749 to (240.99, 147.83, 135.08) mm, rotated rx 180 ry 0 rz 180 deg; joints [-28.7, 14.576, 66.621, 74.383, 29.909, -72.126]
  MoveL 9750 to (240.99, 147.83, 135.08) mm, rotated rx 180 ry 0 rz 180 deg; joints [-28.7, 14.576, 66.621, 74.383, 29.909, -72.126]
  Call Extruder(251.97035)
  MoveL 9751 to (240.95, 148.22, 135.08) mm, rotated rx -180 ry 0 rz 180 deg; joints [-28.737, 14.603, 66.588, 74.395, 29.946, -72.134]
  MoveL 9752 to (240.95, 148.22, 135.08) mm, rotated rx -180 ry 0 rz 180 deg; joints [-28.737, 14.603, 66.588, 74.395, 29.946, -72.134]
  Call Extruder(252.16879)
  MoveL 9753 to (240.9, 148.6, 135.08) mm, rotated rx 180 ry 0 rz 180 deg; joints [-28.774, 14.629, 66.555, 74.408, 29.984, -72.142]
  MoveL 9754 to (240.9, 148.6, 135.08) mm, rotated rx 180 ry 0 rz 180 deg; joints [-28.774, 14.629, 66.555, 74.408, 29.984, -72.142]
  Call Extruder(252.36810)
  MoveL 9755 to (240.86, 148.99, 135.08) mm, rotated rx 180 ry 0 rz 180 deg; joints [-28.812, 14.655, 66.523, 74.42, 30.021, -72.15]
  MoveL 9756 to (240.86, 148.99, 135.08) mm, rotated rx 180 ry 0 rz 180 deg; joints [-28.812, 14.655, 66.523, 74.42, 30.021, -72.15]
  Call Extruder(252.52693)
  MoveL 9757 to (240.81, 149.3, 135.08) mm, rotated rx 180 ry 0 rz 180 deg; joints [-28.842, 14.674, 66.499, 74.431, 30.051, -72.157]
  MoveL 9758 to (240.81, 149.3, 135.08) mm, rotated rx 180 ry 0 rz 180 deg; joints [-28.842, 14.674, 66.499, 74.431, 30.051, -72.157]
  Call Extruder(252.68649)
  MoveL 9759 to (240.76, 149.6, 135.08) mm, rotated rx 180 ry 0 rz 180 deg; joints [-28.872, 14.693, 66.476, 74.442, 30.081, -72.164]
  MoveL 9760 to (240.76, 149.6, 135.08) mm, rotated rx 180 ry 0 rz 180 deg; joints [-28.872, 14.693, 66.476, 74.442, 30.081, -72.164]
  Call Extruder(252.84678)
  MoveL 9761 to (240.71, 149.91, 135.08) mm, rotated rx 180 ry 0 rz 180 deg; joints [-28.902, 14.712, 66.452, 74.452, 30.111, -72.171]
  MoveL 9762 to (240.71, 149.91, 135.08) mm, rotated rx 180 ry 0 rz 180 deg; joints [-28.902, 14.712, 66.452, 74.452, 30.111, -72.171]
  Call Extruder(253.00780)
  MoveL 9763 to (240.66, 150.21, 135.08) mm, rotated rx 180 ry 0 rz 180 deg; joints [-28.932, 14.731, 66.428, 74.463, 30.141, -72.178]
  MoveL 9764 to (240.66, 150.21, 135.08) mm, rotated rx 180 ry 0 rz 180 deg; joints [-28.932, 14.731, 66.428, 74.463, 30.141, -72.178]
  Call Extruder(253.16954)
  MoveL 9765 to (240.61, 150.52, 135.08) mm, rotated rx 180 ry 0 rz 180 deg; joints [-28.962, 14.751, 66.405, 74.474, 30.171, -72.185]
  MoveL 9766 to (240.61, 150.52, 135.08) mm, rotated rx 180 ry 0 rz 180 deg; joints [-28.962, 14.751, 66.405, 74.474, 30.171, -72.185]
  Call Extruder(253.33202)
  MoveL 9767 to (240.57, 150.83, 135.08) mm, rotated rx 180 ry 0 rz 180 deg; joints [-28.993, 14.77, 66.381, 74.485, 30.2, -72.192]
  MoveL 9768 to (240.57, 150.83, 135.08) mm, rotated rx 180 ry 0 rz 180 deg; joints [-28.993, 14.77, 66.381, 74.485, 30.2, -72.192]
  Call Extruder(253.46594)
  MoveL 9769 to (240.52, 151.07, 135.08) mm, rotated rx -180 ry 0 rz 180 deg; joints [-29.017, 14.784, 66.364, 74.494, 30.225, -72.199]
  MoveL 9770 to (240.52, 151.07, 135.08) mm, rotated rx -180 ry 0 rz 180 deg; joints [-29.017, 14.784, 66.364, 74.494, 30.225, -72.199]
  Call Extruder(253.60048)
  MoveL 9771 to (240.47, 151.32, 135.08) mm, rotated rx 180 ry 0 rz 180 deg; joints [-29.043, 14.798, 66.346, 74.504, 30.25, -72.206]
  MoveL 9772 to (240.47, 151.32, 135.08) mm, rotated rx 180 ry 0 rz 180 deg; joints [-29.043, 14.798, 66.346, 74.504, 30.25, -72.206]
  Call Extruder(253.73563)
  MoveL 9773 to (240.42, 151.57, 135.08) mm, rotated rx 180 ry 0 rz 180 deg; joints [-29.067, 14.812, 66.329, 74.513, 30.275, -72.212]
  MoveL 9774 to (240.42, 151.57, 135.08) mm, rotated rx 180 ry 0 rz 180 deg; joints [-29.067, 14.812, 66.329, 74.513, 30.275, -72.212]
  Call Extruder(253.87138)
  MoveL 9775 to (240.37, 151.82, 135.08) mm, rotated rx -180 ry 0 rz 180 deg; joints [-29.092, 14.826, 66.311, 74.523, 30.299, -72.219]
  MoveL 9776 to (240.37, 151.82, 135.08) mm, rotated rx -180 ry 0 rz 180 deg; joints [-29.092, 14.826, 66.311, 74.523, 30.299, -72.219]
  Call Extruder(254.00775)
  MoveL 9777 to (240.32, 152.07, 135.08) mm, rotated rx 180 ry 0 rz 180 deg; joints [-29.117, 14.84, 66.294, 74.532, 30.324, -72.225]
  MoveL 9778 to (240.32, 152.07, 135.08) mm, rotated rx 180 ry 0 rz 180 deg; joints [-29.117, 14.84, 66.294, 74.532, 30.324, -72.225]
  Call Extruder(254.14473)
  MoveL 9779 to (240.27, 152.32, 135.08) mm, rotated rx 180 ry 0 rz 180 deg; joints [-29.142, 14.854, 66.276, 74.542, 30.349, -72.232]
  MoveL 9780 to (240.27, 152.32, 135.08) mm, rotated rx 180 ry 0 rz 180 deg; joints [-29.142, 14.854, 66.276, 74.542, 30.349, -72.232]
  Call Extruder(254.28232)
  MoveL 9781 to (240.22, 152.57, 135.08) mm, rotated rx 180 ry 0 rz -180 deg; joints [-29.167, 14.868, 66.259, 74.551, 30.373, -72.238]
  MoveL 9782 to (240.22, 152.57, 135.08) mm, rotated rx 180 ry 0 rz -180 deg; joints [-29.167, 14.868, 66.259, 74.551, 30.373, -72.238]
  Call Extruder(254.39601)
  MoveL 9783 to (240.17, 152.77, 135.08) mm, rotated rx 180 ry 0 rz 180 deg; joints [-29.188, 14.879, 66.245, 74.559, 30.394, -72.244]
  MoveL 9784 to (240.17, 152.77, 135.08) mm, rotated rx 180 ry 0 rz 180 deg; joints [-29.188, 14.879, 66.245, 74.559, 30.394, -72.244]
  Call Extruder(254.51016)
  MoveL 9785 to (240.13, 152.98, 135.08) mm, rotated rx 180 ry 0 rz 180 deg; joints [-29.209, 14.89, 66.231, 74.567, 30.414, -72.25]
  MoveL 9786 to (240.13, 152.98, 135.08) mm, rotated rx 180 ry 0 rz 180 deg; joints [-29.209, 14.89, 66.231, 74.567, 30.414, -72.25]
  Call Extruder(254.62477)
  MoveL 9787 to (240.08, 153.18, 135.08) mm, rotated rx 180 ry 0 rz 180 deg; joints [-29.229, 14.901, 66.218, 74.575, 30.434, -72.255]
  MoveL 9788 to (240.08, 153.18, 135.08) mm, rotated rx 180 ry 0 rz 180 deg; joints [-29.229, 14.901, 66.218, 74.575, 30.434, -72.255]
  Call Extruder(254.73982)
  MoveL 9789 to (240.04, 153.39, 135.08) mm, rotated rx 180 ry 0 rz 180 deg; joints [-29.25, 14.912, 66.204, 74.583, 30.455, -72.261]
  MoveL 9790 to (240.04, 153.39, 135.08) mm, rotated rx 180 ry 0 rz 180 deg; joints [-29.25, 14.912, 66.204, 74.583, 30.455, -72.261]
  Call Extruder(254.86204)
  MoveL 9791 to (239.98, 153.6, 135.08) mm, rotated rx 180 ry 0 rz 180 deg; joints [-29.272, 14.922, 66.191, 74.593, 30.476, -72.268]
  MoveL 9792 to (239.98, 153.6, 135.08) mm, rotated rx 180 ry 0 rz 180 deg; joints [-29.272, 14.922, 66.191, 74.593, 30.476, -72.268]
  Call Extruder(254.99170)
  MoveL 9793 to (239.92, 153.82, 135.08) mm, rotated rx 180 ry 0 rz -180 deg; joints [-29.296, 14.932, 66.18, 74.603, 30.499, -72.276]
  MoveL 9794 to (239.92, 153.82, 135.08) mm, rotated rx 180 ry 0 rz -180 deg; joints [-29.296, 14.932, 66.18, 74.603, 30.499, -72.276]
  Call Extruder(255.12193)
  MoveL 9795 to (239.85, 154.05, 135.08) mm, rotated rx 180 ry 0 rz 180 deg; joints [-29.319, 14.941, 66.169, 74.614, 30.522, -72.284]
  MoveL 9796 to (239.85, 154.05, 135.08) mm, rotated rx 180 ry 0 rz 180 deg; joints [-29.319, 14.941, 66.169, 74.614, 30.522, -72.284]
  Call Extruder(255.25272)
  MoveL 9797 to (239.78, 154.27, 135.08) mm, rotated rx 180 ry 0 rz 180 deg; joints [-29.343, 14.95, 66.157, 74.624, 30.545, -72.291]
  MoveL 9798 to (239.78, 154.27, 135.08) mm, rotated rx 180 ry 0 rz 180 deg; joints [-29.343, 14.95, 66.157, 74.624, 30.545, -72.291]
  Call Extruder(255.38407)
  MoveL 9799 to (239.71, 154.5, 135.08) mm, rotated rx 180 ry 0 rz 180 deg; joints [-29.366, 14.959, 66.146, 74.634, 30.569, -72.299]
  MoveL 9800 to (239.71, 154.5, 135.08) mm, rotated rx 180 ry 0 rz 180 deg; joints [-29.366, 14.959, 66.146, 74.634, 30.569, -72.299]
  Call Extruder(255.49598)
  MoveL 9801 to (239.65, 154.68, 135.08) mm, rotated rx 180 ry 0 rz 180 deg; joints [-29.386, 14.966, 66.137, 74.644, 30.588, -72.306]
  MoveL 9802 to (239.65, 154.68, 135.08) mm, rotated rx 180 ry 0 rz 180 deg; joints [-29.386, 14.966, 66.137, 74.644, 30.588, -72.306]
  Call Extruder(255.60832)
  MoveL 9803 to (239.59, 154.87, 135.08) mm, rotated rx -180 ry 0 rz 180 deg; joints [-29.406, 14.973, 66.128, 74.653, 30.608, -72.313]
  MoveL 9804 to (239.59, 154.87, 135.08) mm, rotated rx -180 ry 0 rz 180 deg; joints [-29.406, 14.973, 66.128, 74.653, 30.608, -72.313]
  Call Extruder(255.72111)
  MoveL 9805 to (239.53, 155.06, 135.08) mm, rotated rx -180 ry 0 rz 180 deg; joints [-29.426, 14.98, 66.119, 74.662, 30.627, -72.32]
  MoveL 9806 to (239.53, 155.06, 135.08) mm, rotated rx -180 ry 0 rz 180 deg; joints [-29.426, 14.98, 66.119, 74.662, 30.627, -72.32]
  Call Extruder(255.83435)
  MoveL 9807 to (239.47, 155.25, 135.08) mm, rotated rx 180 ry 0 rz -180 deg; joints [-29.446, 14.988, 66.11, 74.671, 30.647, -72.327]
  MoveL 9808 to (239.47, 155.25, 135.08) mm, rotated rx 180 ry 0 rz -180 deg; joints [-29.446, 14.988, 66.11, 74.671, 30.647, -72.327]
  Call Extruder(255.94803)
  MoveL 9809 to (239.41, 155.44, 135.08) mm, rotated rx 180 ry 0 rz 180 deg; joints [-29.466, 14.995, 66.101, 74.68, 30.666, -72.334]
  MoveL 9810 to (239.41, 155.44, 135.08) mm, rotated rx 180 ry 0 rz 180 deg; joints [-29.466, 14.995, 66.101, 74.68, 30.666, -72.334]
  Call Extruder(256.12998)
  MoveL 9811 to (239.29, 155.73, 135.08) mm, rotated rx 180 ry 0 rz -180 deg; joints [-29.499, 15.002, 66.093, 74.696, 30.697, -72.348]
  MoveL 9812 to (239.29, 155.73, 135.08) mm, rotated rx 180 ry 0 rz -180 deg; joints [-29.499, 15.002, 66.093, 74.696, 30.697, -72.348]
  Call Extruder(256.31270)
  MoveL 9813 to (239.16, 156.02, 135.08) mm, rotated rx 180 ry 0 rz 180 deg; joints [-29.531, 15.009, 66.084, 74.713, 30.729, -72.361]
  MoveL 9814 to (239.16, 156.02, 135.08) mm, rotated rx 180 ry 0 rz 180 deg; joints [-29.531, 15.009, 66.084, 74.713, 30.729, -72.361]
  Call Extruder(256.48312)
  MoveL 9815 to (239.05, 156.29, 135.08) mm, rotated rx 180 ry 0 rz 180 deg; joints [-29.561, 15.015, 66.076, 74.728, 30.758, -72.373]
  MoveL 9816 to (239.05, 156.29, 135.08) mm, rotated rx 180 ry 0 rz 180 deg; joints [-29.561, 15.015, 66.076, 74.728, 30.758, -72.373]
  Call Extruder(256.64113)
  MoveL 9817 to (238.94, 156.54, 135.08) mm, rotated rx 180 ry 0 rz 180 deg; joints [-29.589, 15.02, 66.07, 74.743, 30.785, -72.385]
  MoveL 9818 to (238.94, 156.54, 135.08) mm, rotated rx 180 ry 0 rz 180 deg; joints [-29.589, 15.02, 66.07, 74.743, 30.785, -72.385]
  Call Extruder(256.79975)
  MoveL 9819 to (238.84, 156.79, 135.08) mm, rotated rx 180 ry 0 rz 180 deg; joints [-29.617, 15.026, 66.063, 74.757, 30.811, -72.396]
  MoveL 9820 to (238.84, 156.79, 135.08) mm, rotated rx 180 ry 0 rz 180 deg; joints [-29.617, 15.026, 66.063, 74.757, 30.811, -72.396]
  Call Extruder(257.00592)
  MoveL 9821 to (238.66, 157.09, 135.08) mm, rotated rx 180 ry 0 rz 180 deg; joints [-29.653, 15.025, 66.063, 74.778, 30.846, -72.415]
  MoveL 9822 to (238.66, 157.09, 135.08) mm, rotated rx 180 ry 0 rz 180 deg; joints [-29.653, 15.025, 66.063, 74.778, 30.846, -72.415]
  Call Extruder(257.21287)
  MoveL 9823 to (238.49, 157.4, 135.08) mm, rotated rx 180 ry 0 rz -180 deg; joints [-29.689, 15.025, 66.064, 74.8, 30.88, -72.433]
  MoveL 9824 to (238.49, 157.4, 135.08) mm, rotated rx 180 ry 0 rz -180 deg; joints [-29.689, 15.025, 66.064, 74.8, 30.88, -72.433]
  Call Extruder(257.42059)
  MoveL 9825 to (238.31, 157.7, 135.08) mm, rotated rx 180 ry 0 rz 180 deg; joints [-29.725, 15.025, 66.064, 74.821, 30.915, -72.452]
  MoveL 9826 to (238.31, 157.7, 135.08) mm, rotated rx 180 ry 0 rz 180 deg; joints [-29.725, 15.025, 66.064, 74.821, 30.915, -72.452]
  Call Extruder(257.62910)
  MoveL 9827 to (238.13, 158.01, 135.08) mm, rotated rx 180 ry 0 rz 180 deg; joints [-29.761, 15.024, 66.064, 74.842, 30.949, -72.47]
  MoveL 9828 to (238.13, 158.01, 135.08) mm, rotated rx 180 ry 0 rz 180 deg; joints [-29.761, 15.024, 66.064, 74.842, 30.949, -72.47]
  Call Extruder(257.80864)
  MoveL 9829 to (237.96, 158.25, 135.08) mm, rotated rx 180 ry 0 rz 180 deg; joints [-29.792, 15.019, 66.071, 74.863, 30.979, -72.488]
  MoveL 9830 to (237.96, 158.25, 135.08) mm, rotated rx 180 ry 0 rz 180 deg; joints [-29.792, 15.019, 66.071, 74.863, 30.979, -72.488]
  Call Extruder(258.14205)
  MoveL 9831 to (237.63, 158.7, 135.08) mm, rotated rx 180 ry 0 rz 180 deg; joints [-29.849, 15.008, 66.085, 74.9, 31.032, -72.522]
  MoveL 9832 to (237.63, 158.7, 135.08) mm, rotated rx 180 ry 0 rz 180 deg; joints [-29.849, 15.008, 66.085, 74.9, 31.032, -72.522]
  Call Extruder(258.47664)
  MoveL 9833 to (237.3, 159.15, 135.08) mm, rotated rx -180 ry 0 rz -180 deg; joints [-29.907, 14.997, 66.098, 74.938, 31.086, -72.555]
  Call Extruder(259.30463)
  MoveL 9834 to (236.39, 160.19, 135.08) mm, rotated rx 180 ry 0 rz 180 deg; joints [-30.046, 14.948, 66.16, 75.038, 31.216, -72.647]
  Call Extruder(260.13252)
  MoveL 9835 to (235.35, 161.1, 135.08) mm, rotated rx -180 ry 0 rz 180 deg; joints [-30.182, 14.868, 66.259, 75.146, 31.34, -72.749]
  Call Extruder(260.29983)
  MoveL 9836 to (235.13, 161.27, 135.08) mm, rotated rx 180 ry 0 rz -180 deg; joints [-30.208, 14.848, 66.284, 75.169, 31.364, -72.771]
  MoveL 9837 to (235.13, 161.27, 135.08) mm, rotated rx 180 ry 0 rz -180 deg; joints [-30.208, 14.848, 66.284, 75.169, 31.364, -72.771]
  Call Extruder(260.63326)
  MoveL 9838 to (234.68, 161.6, 135.08) mm, rotated rx 180 ry 0 rz 180 deg; joints [-30.261, 14.807, 66.335, 75.215, 31.412, -72.815]
  MoveL 9839 to (234.68, 161.6, 135.08) mm, rotated rx 180 ry 0 rz 180 deg; joints [-30.261, 14.807, 66.335, 75.215, 31.412, -72.815]
  Call Extruder(260.96550)
  MoveL 9840 to (234.22, 161.92, 135.08) mm, rotated rx 180 ry 0 rz 180 deg; joints [-30.314, 14.766, 66.385, 75.26, 31.46, -72.859]
  MoveL 9841 to (234.22, 161.92, 135.08) mm, rotated rx 180 ry 0 rz 180 deg; joints [-30.314, 14.766, 66.385, 75.26, 31.46, -72.859]
  Call Extruder(261.08316)
  MoveL 9842 to (234.05, 162.02, 135.08) mm, rotated rx -180 ry 0 rz 180 deg; joints [-30.331, 14.749, 66.407, 75.277, 31.476, -72.875]
  MoveL 9843 to (234.05, 162.02, 135.08) mm, rotated rx -180 ry 0 rz 180 deg; joints [-30.331, 14.749, 66.407, 75.277, 31.476, -72.875]
  Call Extruder(261.29090)
  MoveL 9844 to (233.75, 162.2, 135.08) mm, rotated rx -180 ry 0 rz 180 deg; joints [-30.363, 14.717, 66.446, 75.306, 31.504, -72.904]
  MoveL 9845 to (233.75, 162.2, 135.08) mm, rotated rx -180 ry 0 rz 180 deg; joints [-30.363, 14.717, 66.446, 75.306, 31.504, -72.904]
  Call Extruder(261.49785)
  MoveL 9846 to (233.45, 162.37, 135.08) mm, rotated rx 180 ry 0 rz 180 deg; joints [-30.394, 14.686, 66.485, 75.336, 31.533, -72.933]
  MoveL 9847 to (233.45, 162.37, 135.08) mm, rotated rx 180 ry 0 rz 180 deg; joints [-30.394, 14.686, 66.485, 75.336, 31.533, -72.933]
  Call Extruder(261.70402)
  MoveL 9848 to (233.14, 162.55, 135.08) mm, rotated rx 180 ry 0 rz 180 deg; joints [-30.426, 14.654, 66.524, 75.366, 31.561, -72.962]
  MoveL 9849 to (233.14, 162.55, 135.08) mm, rotated rx 180 ry 0 rz 180 deg; joints [-30.426, 14.654, 66.524, 75.366, 31.561, -72.962]
  Call Extruder(261.88569)
  MoveL 9850 to (232.87, 162.69, 135.08) mm, rotated rx 180 ry 0 rz -180 deg; joints [-30.453, 14.624, 66.561, 75.392, 31.585, -72.988]
  MoveL 9851 to (232.87, 162.69, 135.08) mm, rotated rx 180 ry 0 rz -180 deg; joints [-30.453, 14.624, 66.561, 75.392, 31.585, -72.988]
  Call Extruder(262.04366)
  MoveL 9852 to (232.62, 162.8, 135.08) mm, rotated rx 180 ry 0 rz -180 deg; joints [-30.476, 14.595, 66.597, 75.416, 31.605, -73.012]
  MoveL 9853 to (232.62, 162.8, 135.08) mm, rotated rx 180 ry 0 rz -180 deg; joints [-30.476, 14.595, 66.597, 75.416, 31.605, -73.012]
  Call Extruder(262.20102)
  MoveL 9854 to (232.37, 162.91, 135.08) mm, rotated rx 180 ry 0 rz 180 deg; joints [-30.498, 14.566, 66.633, 75.439, 31.625, -73.035]
  MoveL 9855 to (232.37, 162.91, 135.08) mm, rotated rx 180 ry 0 rz 180 deg; joints [-30.498, 14.566, 66.633, 75.439, 31.625, -73.035]
  Call Extruder(262.38376)
  MoveL 9856 to (232.07, 163.03, 135.08) mm, rotated rx 180 ry 0 rz 180 deg; joints [-30.524, 14.532, 66.676, 75.466, 31.648, -73.063]
  MoveL 9857 to (232.07, 163.03, 135.08) mm, rotated rx 180 ry 0 rz 180 deg; joints [-30.524, 14.532, 66.676, 75.466, 31.648, -73.063]
  Call Extruder(262.56574)
  MoveL 9858 to (231.78, 163.15, 135.08) mm, rotated rx -180 ry 0 rz 180 deg; joints [-30.551, 14.498, 66.718, 75.494, 31.671, -73.09]
  MoveL 9859 to (231.78, 163.15, 135.08) mm, rotated rx -180 ry 0 rz 180 deg; joints [-30.551, 14.498, 66.718, 75.494, 31.671, -73.09]
  Call Extruder(262.71308)
  MoveL 9860 to (231.54, 163.24, 135.08) mm, rotated rx 180 ry 0 rz 180 deg; joints [-30.571, 14.469, 66.754, 75.516, 31.689, -73.112]
  MoveL 9861 to (231.54, 163.24, 135.08) mm, rotated rx 180 ry 0 rz 180 deg; joints [-30.571, 14.469, 66.754, 75.516, 31.689, -73.112]
  Call Extruder(262.82630)
  MoveL 9862 to (231.35, 163.3, 135.08) mm, rotated rx -180 ry 0 rz 180 deg; joints [-30.587, 14.445, 66.783, 75.533, 31.702, -73.13]
  MoveL 9863 to (231.35, 163.3, 135.08) mm, rotated rx -180 ry 0 rz 180 deg; joints [-30.587, 14.445, 66.783, 75.533, 31.702, -73.13]
  Call Extruder(262.93908)
  MoveL 9864 to (231.17, 163.36, 135.08) mm, rotated rx -180 ry 0 rz 180 deg; joints [-30.602, 14.422, 66.812, 75.55, 31.716, -73.147]
  MoveL 9865 to (231.17, 163.36, 135.08) mm, rotated rx -180 ry 0 rz 180 deg; joints [-30.602, 14.422, 66.812, 75.55, 31.716, -73.147]
  Call Extruder(263.05141)
  MoveL 9866 to (230.98, 163.42, 135.08) mm, rotated rx -180 ry 0 rz 180 deg; joints [-30.618, 14.398, 66.841, 75.567, 31.729, -73.165]
  MoveL 9867 to (230.98, 163.42, 135.08) mm, rotated rx -180 ry 0 rz 180 deg; joints [-30.618, 14.398, 66.841, 75.567, 31.729, -73.165]
  Call Extruder(263.16330)
  MoveL 9868 to (230.79, 163.48, 135.08) mm, rotated rx 180 ry 0 rz 180 deg; joints [-30.633, 14.374, 66.87, 75.585, 31.742, -73.182]
  MoveL 9869 to (230.79, 163.48, 135.08) mm, rotated rx 180 ry 0 rz 180 deg; joints [-30.633, 14.374, 66.87, 75.585, 31.742, -73.182]
  Call Extruder(263.28471)
  MoveL 9870 to (230.58, 163.55, 135.08) mm, rotated rx 180 ry 0 rz 180 deg; joints [-30.65, 14.348, 66.902, 75.603, 31.757, -73.201]
  MoveL 9871 to (230.58, 163.55, 135.08) mm, rotated rx 180 ry 0 rz 180 deg; joints [-30.65, 14.348, 66.902, 75.603, 31.757, -73.201]
  Call Extruder(263.41552)
  MoveL 9872 to (230.36, 163.62, 135.08) mm, rotated rx 180 ry 0 rz -180 deg; joints [-30.668, 14.32, 66.937, 75.623, 31.772, -73.222]
  MoveL 9873 to (230.36, 163.62, 135.08) mm, rotated rx 180 ry 0 rz -180 deg; joints [-30.668, 14.32, 66.937, 75.623, 31.772, -73.222]
  Call Extruder(263.54577)
  MoveL 9874 to (230.14, 163.68, 135.08) mm, rotated rx 180 ry 0 rz 180 deg; joints [-30.685, 14.292, 66.972, 75.644, 31.788, -73.242]
  MoveL 9875 to (230.14, 163.68, 135.08) mm, rotated rx 180 ry 0 rz 180 deg; joints [-30.685, 14.292, 66.972, 75.644, 31.788, -73.242]
  Call Extruder(263.67545)
  MoveL 9876 to (229.91, 163.75, 135.08) mm, rotated rx 180 ry 0 rz 180 deg; joints [-30.703, 14.263, 67.007, 75.664, 31.803, -73.263]
  MoveL 9877 to (229.91, 163.75, 135.08) mm, rotated rx 180 ry 0 rz 180 deg; joints [-30.703, 14.263, 67.007, 75.664, 31.803, -73.263]
  Call Extruder(263.80457)
  MoveL 9878 to (229.69, 163.82, 135.08) mm, rotated rx -180 ry 0 rz 180 deg; joints [-30.721, 14.235, 67.042, 75.684, 31.819, -73.283]
  MoveL 9879 to (229.69, 163.82, 135.08) mm, rotated rx -180 ry 0 rz 180 deg; joints [-30.721, 14.235, 67.042, 75.684, 31.819, -73.283]
  Call Extruder(263.91964)
  MoveL 9880 to (229.48, 163.86, 135.08) mm, rotated rx 180 ry 0 rz 180 deg; joints [-30.736, 14.207, 67.076, 75.702, 31.831, -73.302]
  MoveL 9881 to (229.48, 163.86, 135.08) mm, rotated rx 180 ry 0 rz 180 deg; joints [-30.736, 14.207, 67.076, 75.702, 31.831, -73.302]
  Call Extruder(264.03426)
  MoveL 9882 to (229.28, 163.91, 135.08) mm, rotated rx 180 ry 0 rz 180 deg; joints [-30.751, 14.18, 67.11, 75.72, 31.844, -73.32]
  MoveL 9883 to (229.28, 163.91, 135.08) mm, rotated rx 180 ry 0 rz 180 deg; joints [-30.751, 14.18, 67.11, 75.72, 31.844, -73.32]
  Call Extruder(264.14843)
  MoveL 9884 to (229.08, 163.95, 135.08) mm, rotated rx 180 ry 0 rz 180 deg; joints [-30.766, 14.153, 67.144, 75.738, 31.857, -73.339]
  MoveL 9885 to (229.08, 163.95, 135.08) mm, rotated rx 180 ry 0 rz 180 deg; joints [-30.766, 14.153, 67.144, 75.738, 31.857, -73.339]
  Call Extruder(264.26215)
  MoveL 9886 to (228.87, 164, 135.08) mm, rotated rx 180 ry 0 rz -180 deg; joints [-30.781, 14.125, 67.177, 75.756, 31.87, -73.357]
  MoveL 9887 to (228.87, 164, 135.08) mm, rotated rx 180 ry 0 rz -180 deg; joints [-30.781, 14.125, 67.177, 75.756, 31.87, -73.357]
  Call Extruder(264.38757)
  MoveL 9888 to (228.65, 164.04, 135.08) mm, rotated rx 180 ry 0 rz 180 deg; joints [-30.797, 14.095, 67.215, 75.775, 31.883, -73.378]
  MoveL 9889 to (228.65, 164.04, 135.08) mm, rotated rx 180 ry 0 rz 180 deg; joints [-30.797, 14.095, 67.215, 75.775, 31.883, -73.378]
  Call Extruder(264.52455)
  MoveL 9890 to (228.4, 164.09, 135.08) mm, rotated rx -180 ry 0 rz -180 deg; joints [-30.815, 14.061, 67.256, 75.797, 31.898, -73.4]
  MoveL 9891 to (228.4, 164.09, 135.08) mm, rotated rx -180 ry 0 rz -180 deg; joints [-30.815, 14.061, 67.256, 75.797, 31.898, -73.4]
  Call Extruder(264.66091)
  MoveL 9892 to (228.15, 164.14, 135.08) mm, rotated rx 180 ry 0 rz 180 deg; joints [-30.832, 14.027, 67.298, 75.819, 31.914, -73.422]
  MoveL 9893 to (228.15, 164.14, 135.08) mm, rotated rx 180 ry 0 rz 180 deg; joints [-30.832, 14.027, 67.298, 75.819, 31.914, -73.422]
  Call Extruder(264.79667)
  MoveL 9894 to (227.9, 164.19, 135.08) mm, rotated rx 180 ry 0 rz 180 deg; joints [-30.85, 13.993, 67.34, 75.84, 31.929, -73.445]
  MoveL 9895 to (227.9, 164.19, 135.08) mm, rotated rx 180 ry 0 rz 180 deg; joints [-30.85, 13.993, 67.34, 75.84, 31.929, -73.445]
  Call Extruder(264.93182)
  MoveL 9896 to (227.65, 164.24, 135.08) mm, rotated rx -180 ry 0 rz 180 deg; joints [-30.868, 13.959, 67.381, 75.862, 31.944, -73.467]
  MoveL 9897 to (227.65, 164.24, 135.08) mm, rotated rx -180 ry 0 rz 180 deg; joints [-30.868, 13.959, 67.381, 75.862, 31.944, -73.467]
  Call Extruder(265.06636)
  MoveL 9898 to (227.4, 164.29, 135.08) mm, rotated rx -180 ry 0 rz 180 deg; joints [-30.886, 13.926, 67.422, 75.883, 31.959, -73.489]
  MoveL 9899 to (227.4, 164.29, 135.08) mm, rotated rx -180 ry 0 rz 180 deg; joints [-30.886, 13.926, 67.422, 75.883, 31.959, -73.489]
  Call Extruder(265.20028)
  MoveL 9900 to (227.15, 164.34, 135.08) mm, rotated rx 180 ry 0 rz 180 deg; joints [-30.903, 13.892, 67.464, 75.905, 31.974, -73.511]
  MoveL 9901 to (227.15, 164.34, 135.08) mm, rotated rx 180 ry 0 rz 180 deg; joints [-30.903, 13.892, 67.464, 75.905, 31.974, -73.511]
  Call Extruder(265.34815)
  MoveL 9902 to (226.87, 164.39, 135.08) mm, rotated rx 180 ry 0 rz -180 deg; joints [-30.923, 13.854, 67.51, 75.928, 31.99, -73.536]
  MoveL 9903 to (226.87, 164.39, 135.08) mm, rotated rx 180 ry 0 rz -180 deg; joints [-30.923, 13.854, 67.51, 75.928, 31.99, -73.536]
  Call Extruder(265.50989)
  MoveL 9904 to (226.57, 164.44, 135.08) mm, rotated rx 180 ry 0 rz 180 deg; joints [-30.943, 13.812, 67.562, 75.954, 32.008, -73.562]
  MoveL 9905 to (226.57, 164.44, 135.08) mm, rotated rx 180 ry 0 rz 180 deg; joints [-30.943, 13.812, 67.562, 75.954, 32.008, -73.562]
  Call Extruder(265.67090)
  MoveL 9906 to (226.26, 164.49, 135.08) mm, rotated rx 180 ry 0 rz 180 deg; joints [-30.964, 13.769, 67.614, 75.98, 32.026, -73.589]
  MoveL 9907 to (226.26, 164.49, 135.08) mm, rotated rx 180 ry 0 rz 180 deg; joints [-30.964, 13.769, 67.614, 75.98, 32.026, -73.589]
  Call Extruder(265.83118)
  MoveL 9908 to (225.96, 164.54, 135.08) mm, rotated rx -180 ry 0 rz 180 deg; joints [-30.985, 13.727, 67.666, 76.006, 32.043, -73.616]
  MoveL 9909 to (225.96, 164.54, 135.08) mm, rotated rx -180 ry 0 rz 180 deg; joints [-30.985, 13.727, 67.666, 76.006, 32.043, -73.616]
  Call Extruder(265.99074)
  MoveL 9910 to (225.65, 164.58, 135.08) mm, rotated rx 180 ry 0 rz 180 deg; joints [-31.006, 13.685, 67.718, 76.032, 32.061, -73.643]
  MoveL 9911 to (225.65, 164.58, 135.08) mm, rotated rx 180 ry 0 rz 180 deg; joints [-31.006, 13.685, 67.718, 76.032, 32.061, -73.643]
  Call Extruder(266.14957)
  MoveL 9912 to (225.34, 164.63, 135.08) mm, rotated rx -180 ry 0 rz -180 deg; joints [-31.027, 13.642, 67.769, 76.057, 32.079, -73.669]
  MoveL 9913 to (225.34, 164.63, 135.08) mm, rotated rx -180 ry 0 rz -180 deg; joints [-31.027, 13.642, 67.769, 76.057, 32.079, -73.669]
  Call Extruder(266.32824)
  MoveL 9914 to (225, 164.68, 135.08) mm, rotated rx 180 ry 0 rz 180 deg; joints [-31.049, 13.594, 67.829, 76.086, 32.098, -73.699]
  MoveL 9915 to (225, 164.68, 135.08) mm, rotated rx 180 ry 0 rz 180 deg; joints [-31.049, 13.594, 67.829, 76.086, 32.098, -73.699]
  Call Extruder(266.52668)
  MoveL 9916 to (224.61, 164.73, 135.08) mm, rotated rx 180 ry 0 rz -180 deg; joints [-31.074, 13.539, 67.896, 76.118, 32.119, -73.733]
  MoveL 9917 to (224.61, 164.73, 135.08) mm, rotated rx 180 ry 0 rz -180 deg; joints [-31.074, 13.539, 67.896, 76.118, 32.119, -73.733]
  Call Extruder(266.72426)
  MoveL 9918 to (224.22, 164.77, 135.08) mm, rotated rx 180 ry 0 rz -180 deg; joints [-31.1, 13.484, 67.963, 76.15, 32.14, -73.766]
  MoveL 9919 to (224.22, 164.77, 135.08) mm, rotated rx 180 ry 0 rz -180 deg; joints [-31.1, 13.484, 67.963, 76.15, 32.14, -73.766]
  Call Extruder(266.92097)
  MoveL 9920 to (223.84, 164.82, 135.08) mm, rotated rx 180 ry 0 rz 180 deg; joints [-31.125, 13.429, 68.03, 76.182, 32.161, -73.799]
  MoveL 9921 to (223.84, 164.82, 135.08) mm, rotated rx 180 ry 0 rz 180 deg; joints [-31.125, 13.429, 68.03, 76.182, 32.161, -73.799]
  Call Extruder(267.11680)
  MoveL 9922 to (223.45, 164.86, 135.08) mm, rotated rx 180 ry 0 rz -180 deg; joints [-31.15, 13.374, 68.096, 76.213, 32.183, -73.832]
  MoveL 9923 to (223.45, 164.86, 135.08) mm, rotated rx 180 ry 0 rz -180 deg; joints [-31.15, 13.374, 68.096, 76.213, 32.183, -73.832]
  Call Extruder(267.41216)
  MoveL 9924 to (222.86, 164.91, 135.08) mm, rotated rx -180 ry 0 rz 180 deg; joints [-31.186, 13.289, 68.2, 76.261, 32.213, -73.882]
  MoveL 9925 to (222.86, 164.91, 135.08) mm, rotated rx -180 ry 0 rz 180 deg; joints [-31.186, 13.289, 68.2, 76.261, 32.213, -73.882]
  Call Extruder(267.70619)
  MoveL 9926 to (222.27, 164.96, 135.08) mm, rotated rx 180 ry 0 rz -180 deg; joints [-31.222, 13.204, 68.304, 76.308, 32.243, -73.931]
  MoveL 9927 to (222.27, 164.96, 135.08) mm, rotated rx 180 ry 0 rz -180 deg; joints [-31.222, 13.204, 68.304, 76.308, 32.243, -73.931]
  Call Extruder(267.99889)
  MoveL 9928 to (221.68, 165, 135.08) mm, rotated rx -180 ry 0 rz 180 deg; joints [-31.258, 13.119, 68.407, 76.355, 32.274, -73.98]
  MoveL 9929 to (221.68, 165, 135.08) mm, rotated rx -180 ry 0 rz 180 deg; joints [-31.258, 13.119, 68.407, 76.355, 32.274, -73.98]
  Call Extruder(268.57233)
  MoveL 9930 to (220.52, 165.05, 135.08) mm, rotated rx -180 ry 0 rz 180 deg; joints [-31.326, 12.948, 68.615, 76.445, 32.331, -74.076]
  MoveL 9931 to (220.52, 165.05, 135.08) mm, rotated rx -180 ry 0 rz 180 deg; joints [-31.326, 12.948, 68.615, 76.445, 32.331, -74.076]
  Call Extruder(269.28634)
  MoveL 9932 to (219.06, 165.09, 135.08) mm, rotated rx 180 ry 0 rz 180 deg; joints [-31.409, 12.732, 68.875, 76.557, 32.4, -74.194]
  Call Extruder(386.13307)
  MoveL 9933 to (-19.06, 165.09, 135.08) mm, rotated rx 180 ry 0 rz 180 deg; joints [-51.475, -15.737, 96.647, 82.831, 52.046, -78.442]
  Call Extruder(386.56168)
  MoveL 9934 to (-19.94, 165.07, 135.08) mm, rotated rx 180 ry 0 rz 180 deg; joints [-51.582, -15.819, 96.708, 82.842, 52.153, -78.432]
  MoveL 9935 to (-19.94, 165.07, 135.08) mm, rotated rx 180 ry 0 rz 180 deg; joints [-51.582, -15.819, 96.708, 82.842, 52.153, -78.432]
  Call Extruder(387.13513)
  MoveL 9936 to (-21.1, 165.03, 135.08) mm, rotated rx 180 ry 0 rz 180 deg; joints [-51.722, -15.93, 96.79, 82.855, 52.294, -78.418]
  MoveL 9937 to (-21.1, 165.03, 135.08) mm, rotated rx 180 ry 0 rz 180 deg; joints [-51.722, -15.93, 96.79, 82.855, 52.294, -78.418]
  Call Extruder(387.56943)
  MoveL 9938 to (-21.97, 164.98, 135.08) mm, rotated rx -180 ry 0 rz 180 deg; joints [-51.827, -16.015, 96.853, 82.865, 52.4, -78.406]
  MoveL 9939 to (-21.97, 164.98, 135.08) mm, rotated rx -180 ry 0 rz 180 deg; joints [-51.827, -16.015, 96.853, 82.865, 52.4, -78.406]
  Call Extruder(387.86345)
  MoveL 9940 to (-22.56, 164.93, 135.08) mm, rotated rx 180 ry 0 rz -180 deg; joints [-51.897, -16.074, 96.896, 82.871, 52.469, -78.398]
  MoveL 9941 to (-22.56, 164.93, 135.08) mm, rotated rx 180 ry 0 rz -180 deg; joints [-51.897, -16.074, 96.896, 82.871, 52.469, -78.398]
  Call Extruder(388.15881)
  MoveL 9942 to (-23.15, 164.89, 135.08) mm, rotated rx -180 ry 0 rz 180 deg; joints [-51.966, -16.132, 96.94, 82.877, 52.539, -78.389]
  MoveL 9943 to (-23.15, 164.89, 135.08) mm, rotated rx -180 ry 0 rz 180 deg; joints [-51.966, -16.132, 96.94, 82.877, 52.539, -78.389]
  Call Extruder(388.40503)
  MoveL 9944 to (-23.64, 164.84, 135.08) mm, rotated rx -180 ry 0 rz 180 deg; joints [-52.023, -16.181, 96.976, 82.881, 52.597, -78.382]
  MoveL 9945 to (-23.64, 164.84, 135.08) mm, rotated rx -180 ry 0 rz 180 deg; joints [-52.023, -16.181, 96.976, 82.881, 52.597, -78.382]
  Call Extruder(388.60173)
  MoveL 9946 to (-24.03, 164.79, 135.08) mm, rotated rx 180 ry 0 rz 180 deg; joints [-52.067, -16.222, 97.005, 82.885, 52.641, -78.375]
  MoveL 9947 to (-24.03, 164.79, 135.08) mm, rotated rx 180 ry 0 rz 180 deg; joints [-52.067, -16.222, 97.005, 82.885, 52.641, -78.375]
  Call Extruder(388.79931)
  MoveL 9948 to (-24.42, 164.75, 135.08) mm, rotated rx 180 ry 0 rz -180 deg; joints [-52.112, -16.262, 97.035, 82.888, 52.686, -78.369]
  MoveL 9949 to (-24.42, 164.75, 135.08) mm, rotated rx 180 ry 0 rz -180 deg; joints [-52.112, -16.262, 97.035, 82.888, 52.686, -78.369]
  Call Extruder(388.99775)
  MoveL 9950 to (-24.8, 164.7, 135.08) mm, rotated rx -180 ry 0 rz 180 deg; joints [-52.156, -16.302, 97.065, 82.891, 52.731, -78.363]
  MoveL 9951 to (-24.8, 164.7, 135.08) mm, rotated rx -180 ry 0 rz 180 deg; joints [-52.156, -16.302, 97.065, 82.891, 52.731, -78.363]
  Call Extruder(389.19706)
  MoveL 9952 to (-25.19, 164.66, 135.08) mm, rotated rx 180 ry 0 rz 180 deg; joints [-52.2, -16.342, 97.094, 82.894, 52.776, -78.356]
  MoveL 9953 to (-25.19, 164.66, 135.08) mm, rotated rx 180 ry 0 rz 180 deg; joints [-52.2, -16.342, 97.094, 82.894, 52.776, -78.356]
  Call Extruder(389.35589)
  MoveL 9954 to (-25.5, 164.61, 135.08) mm, rotated rx 180 ry 0 rz 180 deg; joints [-52.235, -16.375, 97.118, 82.896, 52.81, -78.35]
  MoveL 9955 to (-25.5, 164.61, 135.08) mm, rotated rx 180 ry 0 rz 180 deg; joints [-52.235, -16.375, 97.118, 82.896, 52.81, -78.35]
  Call Extruder(389.51545)
  MoveL 9956 to (-25.8, 164.56, 135.08) mm, rotated rx 180 ry 0 rz 180 deg; joints [-52.269, -16.408, 97.142, 82.898, 52.845, -78.344]
  MoveL 9957 to (-25.8, 164.56, 135.08) mm, rotated rx 180 ry 0 rz 180 deg; joints [-52.269, -16.408, 97.142, 82.898, 52.845, -78.344]
  Call Extruder(389.67574)
  MoveL 9958 to (-26.11, 164.51, 135.08) mm, rotated rx 180 ry 0 rz -180 deg; joints [-52.303, -16.441, 97.166, 82.9, 52.879, -78.339]
  MoveL 9959 to (-26.11, 164.51, 135.08) mm, rotated rx 180 ry 0 rz -180 deg; joints [-52.303, -16.441, 97.166, 82.9, 52.879, -78.339]
  Call Extruder(389.83676)
  MoveL 9960 to (-26.41, 164.46, 135.08) mm, rotated rx -180 ry 0 rz 180 deg; joints [-52.337, -16.474, 97.191, 82.902, 52.914, -78.333]
  MoveL 9961 to (-26.41, 164.46, 135.08) mm, rotated rx -180 ry 0 rz 180 deg; joints [-52.337, -16.474, 97.191, 82.902, 52.914, -78.333]
  Call Extruder(389.99850)
  MoveL 9962 to (-26.72, 164.41, 135.08) mm, rotated rx 180 ry 0 rz -180 deg; joints [-52.371, -16.507, 97.215, 82.904, 52.948, -78.327]
  MoveL 9963 to (-26.72, 164.41, 135.08) mm, rotated rx 180 ry 0 rz -180 deg; joints [-52.371, -16.507, 97.215, 82.904, 52.948, -78.327]
  Call Extruder(390.16097)
  MoveL 9964 to (-27.03, 164.37, 135.08) mm, rotated rx 180 ry 0 rz 180 deg; joints [-52.405, -16.54, 97.239, 82.906, 52.983, -78.321]
  MoveL 9965 to (-27.03, 164.37, 135.08) mm, rotated rx 180 ry 0 rz 180 deg; joints [-52.405, -16.54, 97.239, 82.906, 52.983, -78.321]
  Call Extruder(390.29490)
  MoveL 9966 to (-27.27, 164.32, 135.08) mm, rotated rx -180 ry 0 rz -180 deg; joints [-52.432, -16.568, 97.259, 82.907, 53.01, -78.316]
  MoveL 9967 to (-27.27, 164.32, 135.08) mm, rotated rx -180 ry 0 rz -180 deg; joints [-52.432, -16.568, 97.259, 82.907, 53.01, -78.316]
  Call Extruder(390.42943)
  MoveL 9968 to (-27.52, 164.27, 135.08) mm, rotated rx 180 ry 0 rz 180 deg; joints [-52.459, -16.596, 97.28, 82.909, 53.037, -78.311]
  MoveL 9969 to (-27.52, 164.27, 135.08) mm, rotated rx 180 ry 0 rz 180 deg; joints [-52.459, -16.596, 97.28, 82.909, 53.037, -78.311]
  Call Extruder(390.56458)
  MoveL 9970 to (-27.77, 164.22, 135.08) mm, rotated rx 180 ry 0 rz 180 deg; joints [-52.486, -16.624, 97.3, 82.91, 53.065, -78.305]
  MoveL 9971 to (-27.77, 164.22, 135.08) mm, rotated rx 180 ry 0 rz 180 deg; joints [-52.486, -16.624, 97.3, 82.91, 53.065, -78.305]
  Call Extruder(390.70034)
  MoveL 9972 to (-28.02, 164.17, 135.08) mm, rotated rx 180 ry 0 rz -180 deg; joints [-52.513, -16.652, 97.32, 82.911, 53.092, -78.3]
  MoveL 9973 to (-28.02, 164.17, 135.08) mm, rotated rx 180 ry 0 rz -180 deg; joints [-52.513, -16.652, 97.32, 82.911, 53.092, -78.3]
  Call Extruder(390.83670)
  MoveL 9974 to (-28.27, 164.12, 135.08) mm, rotated rx -180 ry 0 rz 180 deg; joints [-52.54, -16.68, 97.341, 82.912, 53.119, -78.295]
  MoveL 9975 to (-28.27, 164.12, 135.08) mm, rotated rx -180 ry 0 rz 180 deg; joints [-52.54, -16.68, 97.341, 82.912, 53.119, -78.295]
  Call Extruder(390.97368)
  MoveL 9976 to (-28.52, 164.07, 135.08) mm, rotated rx 180 ry 0 rz 180 deg; joints [-52.567, -16.708, 97.361, 82.913, 53.147, -78.289]
  MoveL 9977 to (-28.52, 164.07, 135.08) mm, rotated rx 180 ry 0 rz 180 deg; joints [-52.567, -16.708, 97.361, 82.913, 53.147, -78.289]
  Call Extruder(391.11127)
  MoveL 9978 to (-28.77, 164.02, 135.08) mm, rotated rx 180 ry 0 rz 180 deg; joints [-52.594, -16.736, 97.381, 82.915, 53.174, -78.284]
  MoveL 9979 to (-28.77, 164.02, 135.08) mm, rotated rx 180 ry 0 rz 180 deg; joints [-52.594, -16.736, 97.381, 82.915, 53.174, -78.284]
  Call Extruder(391.22498)
  MoveL 9980 to (-28.97, 163.97, 135.08) mm, rotated rx -180 ry 0 rz 180 deg; joints [-52.616, -16.759, 97.398, 82.915, 53.197, -78.28]
  MoveL 9981 to (-28.97, 163.97, 135.08) mm, rotated rx -180 ry 0 rz 180 deg; joints [-52.616, -16.759, 97.398, 82.915, 53.197, -78.28]
  Call Extruder(391.33915)
  MoveL 9982 to (-29.18, 163.93, 135.08) mm, rotated rx -180 ry 0 rz 180 deg; joints [-52.638, -16.782, 97.415, 82.916, 53.219, -78.275]
  MoveL 9983 to (-29.18, 163.93, 135.08) mm, rotated rx -180 ry 0 rz 180 deg; joints [-52.638, -16.782, 97.415, 82.916, 53.219, -78.275]
  Call Extruder(391.45377)
  MoveL 9984 to (-29.38, 163.88, 135.08) mm, rotated rx 180 ry 0 rz 180 deg; joints [-52.659, -16.806, 97.432, 82.917, 53.241, -78.27]
  MoveL 9985 to (-29.38, 163.88, 135.08) mm, rotated rx 180 ry 0 rz 180 deg; joints [-52.659, -16.806, 97.432, 82.917, 53.241, -78.27]
  Call Extruder(391.56884)
  MoveL 9986 to (-29.59, 163.84, 135.08) mm, rotated rx -180 ry 0 rz 180 deg; joints [-52.681, -16.829, 97.449, 82.918, 53.263, -78.266]
  MoveL 9987 to (-29.59, 163.84, 135.08) mm, rotated rx -180 ry 0 rz 180 deg; joints [-52.681, -16.829, 97.449, 82.918, 53.263, -78.266]
  Call Extruder(391.69108)
  MoveL 9988 to (-29.8, 163.78, 135.08) mm, rotated rx 180 ry 0 rz 180 deg; joints [-52.703, -16.854, 97.467, 82.918, 53.285, -78.261]
  MoveL 9989 to (-29.8, 163.78, 135.08) mm, rotated rx 180 ry 0 rz 180 deg; joints [-52.703, -16.854, 97.467, 82.918, 53.285, -78.261]
  Call Extruder(391.82075)
  MoveL 9990 to (-30.02, 163.72, 135.08) mm, rotated rx -180 ry 0 rz 180 deg; joints [-52.726, -16.882, 97.487, 82.918, 53.308, -78.254]
  MoveL 9991 to (-30.02, 163.72, 135.08) mm, rotated rx -180 ry 0 rz 180 deg; joints [-52.726, -16.882, 97.487, 82.918, 53.308, -78.254]
  Call Extruder(391.95100)
  MoveL 9992 to (-30.25, 163.65, 135.08) mm, rotated rx 180 ry 0 rz 180 deg; joints [-52.748, -16.91, 97.508, 82.918, 53.331, -78.248]
  MoveL 9993 to (-30.25, 163.65, 135.08) mm, rotated rx 180 ry 0 rz 180 deg; joints [-52.748, -16.91, 97.508, 82.918, 53.331, -78.248]
  Call Extruder(392.08180)
  MoveL 9994 to (-30.47, 163.58, 135.08) mm, rotated rx 180 ry 0 rz 180 deg; joints [-52.77, -16.937, 97.528, 82.918, 53.354, -78.242]
  MoveL 9995 to (-30.47, 163.58, 135.08) mm, rotated rx 180 ry 0 rz 180 deg; joints [-52.77, -16.937, 97.528, 82.918, 53.354, -78.242]
  Call Extruder(392.21318)
  MoveL 9996 to (-30.7, 163.51, 135.08) mm, rotated rx 180 ry 0 rz 180 deg; joints [-52.792, -16.965, 97.548, 82.918, 53.376, -78.236]
  MoveL 9997 to (-30.7, 163.51, 135.08) mm, rotated rx 180 ry 0 rz 180 deg; joints [-52.792, -16.965, 97.548, 82.918, 53.376, -78.236]
  Call Extruder(392.32507)
  MoveL 9998 to (-30.88, 163.45, 135.08) mm, rotated rx -180 ry 0 rz 180 deg; joints [-52.81, -16.989, 97.565, 82.918, 53.395, -78.231]
  MoveL 9999 to (-30.88, 163.45, 135.08) mm, rotated rx -180 ry 0 rz 180 deg; joints [-52.81, -16.989, 97.565, 82.918, 53.395, -78.231]
  Call Extruder(392.43740)
  MoveL 10000 to (-31.07, 163.39, 135.08) mm, rotated rx -180 ry 0 rz 180 deg; joints [-52.829, -17.013, 97.582, 82.918, 53.414, -78.225]
  MoveL 10001 to (-31.07, 163.39, 135.08) mm, rotated rx -180 ry 0 rz 180 deg; joints [-52.829, -17.013, 97.582, 82.918, 53.414, -78.225]
  Call Extruder(392.55019)
  MoveL 10002 to (-31.26, 163.33, 135.08) mm, rotated rx -180 ry 0 rz 180 deg; joints [-52.847, -17.036, 97.599, 82.918, 53.433, -78.22]
  MoveL 10003 to (-31.26, 163.33, 135.08) mm, rotated rx -180 ry 0 rz 180 deg; joints [-52.847, -17.036, 97.599, 82.918, 53.433, -78.22]
  Call Extruder(392.66341)
  MoveL 10004 to (-31.45, 163.27, 135.08) mm, rotated rx 180 ry 0 rz 180 deg; joints [-52.866, -17.06, 97.616, 82.917, 53.451, -78.215]
  MoveL 10005 to (-31.45, 163.27, 135.08) mm, rotated rx 180 ry 0 rz 180 deg; joints [-52.866, -17.06, 97.616, 82.917, 53.451, -78.215]
  Call Extruder(392.77708)
  MoveL 10006 to (-31.64, 163.21, 135.08) mm, rotated rx 180 ry 0 rz 180 deg; joints [-52.884, -17.084, 97.633, 82.917, 53.47, -78.209]
  MoveL 10007 to (-31.64, 163.21, 135.08) mm, rotated rx 180 ry 0 rz 180 deg; joints [-52.884, -17.084, 97.633, 82.917, 53.47, -78.209]
  Call Extruder(392.95906)
  MoveL 10008 to (-31.93, 163.09, 135.08) mm, rotated rx 180 ry 0 rz 180 deg; joints [-52.91, -17.124, 97.662, 82.916, 53.497, -78.2]
  MoveL 10009 to (-31.93, 163.09, 135.08) mm, rotated rx 180 ry 0 rz 180 deg; joints [-52.91, -17.124, 97.662, 82.916, 53.497, -78.2]
  Call Extruder(393.14179)
  MoveL 10010 to (-32.22, 162.97, 135.08) mm, rotated rx 180 ry 0 rz -180 deg; joints [-52.936, -17.163, 97.691, 82.914, 53.524, -78.19]
  MoveL 10011 to (-32.22, 162.97, 135.08) mm, rotated rx 180 ry 0 rz -180 deg; joints [-52.936, -17.163, 97.691, 82.914, 53.524, -78.19]
  Call Extruder(393.31221)
  MoveL 10012 to (-32.49, 162.85, 135.08) mm, rotated rx -180 ry 0 rz 180 deg; joints [-52.96, -17.2, 97.717, 82.913, 53.549, -78.181]
  MoveL 10013 to (-32.49, 162.85, 135.08) mm, rotated rx -180 ry 0 rz 180 deg; joints [-52.96, -17.2, 97.717, 82.913, 53.549, -78.181]
  Call Extruder(393.47018)
  MoveL 10014 to (-32.74, 162.74, 135.08) mm, rotated rx 180 ry 0 rz 180 deg; joints [-52.982, -17.235, 97.742, 82.911, 53.571, -78.172]
  MoveL 10015 to (-32.74, 162.74, 135.08) mm, rotated rx 180 ry 0 rz 180 deg; joints [-52.982, -17.235, 97.742, 82.911, 53.571, -78.172]
  Call Extruder(393.62876)
  MoveL 10016 to (-32.99, 162.64, 135.08) mm, rotated rx 180 ry 0 rz -180 deg; joints [-53.004, -17.269, 97.767, 82.91, 53.594, -78.163]
  MoveL 10017 to (-32.99, 162.64, 135.08) mm, rotated rx 180 ry 0 rz -180 deg; joints [-53.004, -17.269, 97.767, 82.91, 53.594, -78.163]
  Call Extruder(393.83493)
  MoveL 10018 to (-33.29, 162.46, 135.08) mm, rotated rx 180 ry 0 rz -180 deg; joints [-53.026, -17.316, 97.801, 82.906, 53.618, -78.15]
  MoveL 10019 to (-33.29, 162.46, 135.08) mm, rotated rx 180 ry 0 rz -180 deg; joints [-53.026, -17.316, 97.801, 82.906, 53.618, -78.15]
  Call Extruder(394.04187)
  MoveL 10020 to (-33.6, 162.29, 135.08) mm, rotated rx 180 ry 0 rz 180 deg; joints [-53.049, -17.364, 97.835, 82.902, 53.641, -78.137]
  MoveL 10021 to (-33.6, 162.29, 135.08) mm, rotated rx 180 ry 0 rz 180 deg; joints [-53.049, -17.364, 97.835, 82.902, 53.641, -78.137]
  Call Extruder(394.24959)
  MoveL 10022 to (-33.9, 162.11, 135.08) mm, rotated rx -180 ry 0 rz 180 deg; joints [-53.071, -17.411, 97.868, 82.898, 53.665, -78.124]
  MoveL 10023 to (-33.9, 162.11, 135.08) mm, rotated rx -180 ry 0 rz 180 deg; joints [-53.071, -17.411, 97.868, 82.898, 53.665, -78.124]
  Call Extruder(394.45809)
  MoveL 10024 to (-34.21, 161.94, 135.08) mm, rotated rx 180 ry 0 rz 180 deg; joints [-53.094, -17.458, 97.902, 82.894, 53.689, -78.111]
  MoveL 10025 to (-34.21, 161.94, 135.08) mm, rotated rx 180 ry 0 rz 180 deg; joints [-53.094, -17.458, 97.902, 82.894, 53.689, -78.111]
  Call Extruder(394.63764)
  MoveL 10026 to (-34.45, 161.76, 135.08) mm, rotated rx 180 ry 0 rz 180 deg; joints [-53.109, -17.5, 97.932, 82.889, 53.704, -78.099]
  MoveL 10027 to (-34.45, 161.76, 135.08) mm, rotated rx 180 ry 0 rz 180 deg; joints [-53.109, -17.5, 97.932, 82.889, 53.704, -78.099]
  Call Extruder(394.97107)
  MoveL 10028 to (-34.9, 161.43, 135.08) mm, rotated rx 180 ry 0 rz 180 deg; joints [-53.135, -17.578, 97.988, 82.879, 53.734, -78.075]
  MoveL 10029 to (-34.9, 161.43, 135.08) mm, rotated rx 180 ry 0 rz 180 deg; joints [-53.135, -17.578, 97.988, 82.879, 53.734, -78.075]
  Call Extruder(395.30569)
  MoveL 10030 to (-35.35, 161.1, 135.08) mm, rotated rx 180 ry 0 rz -180 deg; joints [-53.163, -17.656, 98.043, 82.87, 53.763, -78.052]
  Call Extruder(396.13360)
  MoveL 10031 to (-36.39, 160.19, 135.08) mm, rotated rx 180 ry 0 rz 180 deg; joints [-53.209, -17.853, 98.183, 82.84, 53.816, -77.989]
  Call Extruder(396.96153)
  MoveL 10032 to (-37.3, 159.15, 135.08) mm, rotated rx 180 ry 0 rz -180 deg; joints [-53.227, -18.053, 98.325, 82.803, 53.841, -77.919]
  Call Extruder(397.12884)
  MoveL 10033 to (-37.47, 158.93, 135.08) mm, rotated rx 180 ry 0 rz -180 deg; joints [-53.227, -18.094, 98.354, 82.794, 53.842, -77.904]
  MoveL 10034 to (-37.47, 158.93, 135.08) mm, rotated rx 180 ry 0 rz -180 deg; joints [-53.227, -18.094, 98.354, 82.794, 53.842, -77.904]
  Call Extruder(397.46227)
  MoveL 10035 to (-37.8, 158.48, 135.08) mm, rotated rx 180 ry 0 rz 180 deg; joints [-53.226, -18.175, 98.411, 82.776, 53.843, -77.875]
  MoveL 10036 to (-37.8, 158.48, 135.08) mm, rotated rx 180 ry 0 rz 180 deg; joints [-53.226, -18.175, 98.411, 82.776, 53.843, -77.875]
  Call Extruder(397.53291)
  MoveL 10037 to (-37.87, 158.38, 135.08) mm, rotated rx 180 ry 0 rz 180 deg; joints [-53.225, -18.192, 98.423, 82.772, 53.844, -77.868]
  Set speed (130.0 mm/s)
  MoveL 10038 to (-39.48, 155.51, 135.08) mm, rotated rx 180 ry 0 rz 180 deg; joints [-53.153, -18.668, 98.755, 82.649, 53.792, -77.681]
  MoveL 10039 to (-39.48, 155.51, 144.49) mm, rotated rx -180 ry 0 rz 180 deg; joints [-53.153, -19.217, 100.535, 83.546, 53.644, -79.196]
  MoveL 10040 to (-38.84, 156.79, 144.49) mm, rotated rx -180 ry 0 rz 180 deg; joints [-53.196, -19.011, 100.392, 83.603, 53.679, -79.281]
  Set speed (30.0 mm/s)
  MoveL 10041 to (-38.84, 156.79, 144.49) mm, rotated rx -180 ry 0 rz 180 deg; joints [-53.196, -19.011, 100.392, 83.603, 53.679, -79.281]
  Call Extruder(397.61221)
  MoveL 10042 to (-38.89, 156.67, 144.49) mm, rotated rx 180 ry 0 rz 180 deg; joints [-53.191, -19.03, 100.406, 83.597, 53.674, -79.273]
  MoveL 10043 to (-38.89, 156.67, 144.49) mm, rotated rx 180 ry 0 rz 180 deg; joints [-53.191, -19.03, 100.406, 83.597, 53.674, -79.273]
  Call Extruder(397.77019)
  MoveL 10044 to (-39, 156.42, 144.49) mm, rotated rx 180 ry 0 rz 180 deg; joints [-53.18, -19.069, 100.432, 83.586, 53.665, -79.257]
  MoveL 10045 to (-39, 156.42, 144.49) mm, rotated rx 180 ry 0 rz 180 deg; joints [-53.18, -19.069, 100.432, 83.586, 53.665, -79.257]
  Call Extruder(397.92758)
  MoveL 10046 to (-39.11, 156.17, 144.49) mm, rotated rx -180 ry 0 rz 180 deg; joints [-53.17, -19.107, 100.459, 83.575, 53.656, -79.241]
  MoveL 10047 to (-39.11, 156.17, 144.49) mm, rotated rx -180 ry 0 rz 180 deg; joints [-53.17, -19.107, 100.459, 83.575, 53.656, -79.241]
  Call Extruder(398.11030)
  MoveL 10048 to (-39.22, 155.88, 144.49) mm, rotated rx 180 ry 0 rz 180 deg; joints [-53.156, -19.152, 100.49, 83.562, 53.645, -79.222]
  MoveL 10049 to (-39.22, 155.88, 144.49) mm, rotated rx 180 ry 0 rz 180 deg; joints [-53.156, -19.152, 100.49, 83.562, 53.645, -79.222]
  Call Extruder(398.29226)
  MoveL 10050 to (-39.35, 155.58, 144.49) mm, rotated rx -180 ry 0 rz 180 deg; joints [-53.143, -19.197, 100.521, 83.548, 53.633, -79.203]
  MoveL 10051 to (-39.35, 155.58, 144.49) mm, rotated rx -180 ry 0 rz 180 deg; joints [-53.143, -19.197, 100.521, 83.548, 53.633, -79.203]
  Call Extruder(398.43959)
  MoveL 10052 to (-39.44, 155.34, 144.49) mm, rotated rx 180 ry 0 rz 180 deg; joints [-53.131, -19.233, 100.546, 83.537, 53.623, -79.187]
  MoveL 10053 to (-39.44, 155.34, 144.49) mm, rotated rx 180 ry 0 rz 180 deg; joints [-53.131, -19.233, 100.546, 83.537, 53.623, -79.187]
  Call Extruder(398.55283)
  MoveL 10054 to (-39.5, 155.15, 144.49) mm, rotated rx 180 ry 0 rz -180 deg; joints [-53.121, -19.261, 100.565, 83.529, 53.613, -79.175]
  MoveL 10055 to (-39.5, 155.15, 144.49) mm, rotated rx 180 ry 0 rz -180 deg; joints [-53.121, -19.261, 100.565, 83.529, 53.613, -79.175]
  Call Extruder(398.66562)
  MoveL 10056 to (-39.56, 154.97, 144.49) mm, rotated rx -180 ry 0 rz 180 deg; joints [-53.11, -19.288, 100.584, 83.52, 53.604, -79.163]
  MoveL 10057 to (-39.56, 154.97, 144.49) mm, rotated rx -180 ry 0 rz 180 deg; joints [-53.11, -19.288, 100.584, 83.52, 53.604, -79.163]
  Call Extruder(398.77796)
  MoveL 10058 to (-39.62, 154.78, 144.49) mm, rotated rx 180 ry 0 rz 180 deg; joints [-53.099, -19.315, 100.603, 83.511, 53.594, -79.151]
  MoveL 10059 to (-39.62, 154.78, 144.49) mm, rotated rx 180 ry 0 rz 180 deg; joints [-53.099, -19.315, 100.603, 83.511, 53.594, -79.151]
  Call Extruder(398.88986)
  MoveL 10060 to (-39.68, 154.59, 144.49) mm, rotated rx 180 ry 0 rz -180 deg; joints [-53.088, -19.343, 100.621, 83.502, 53.584, -79.139]
  MoveL 10061 to (-39.68, 154.59, 144.49) mm, rotated rx 180 ry 0 rz -180 deg; joints [-53.088, -19.343, 100.621, 83.502, 53.584, -79.139]
  Call Extruder(399.01126)
  MoveL 10062 to (-39.75, 154.38, 144.49) mm, rotated rx 180 ry 0 rz 180 deg; joints [-53.076, -19.373, 100.642, 83.493, 53.574, -79.126]
  MoveL 10063 to (-39.75, 154.38, 144.49) mm, rotated rx 180 ry 0 rz 180 deg; joints [-53.076, -19.373, 100.642, 83.493, 53.574, -79.126]
  Call Extruder(399.14206)
  MoveL 10064 to (-39.81, 154.16, 144.49) mm, rotated rx 180 ry 0 rz 180 deg; joints [-53.063, -19.405, 100.664, 83.482, 53.561, -79.112]
  MoveL 10065 to (-39.81, 154.16, 144.49) mm, rotated rx 180 ry 0 rz 180 deg; joints [-53.063, -19.405, 100.664, 83.482, 53.561, -79.112]
  Call Extruder(399.27229)
  MoveL 10066 to (-39.88, 153.94, 144.49) mm, rotated rx 180 ry 0 rz 180 deg; joints [-53.049, -19.437, 100.686, 83.471, 53.549, -79.097]
  MoveL 10067 to (-39.88, 153.94, 144.49) mm, rotated rx 180 ry 0 rz 180 deg; joints [-53.049, -19.437, 100.686, 83.471, 53.549, -79.097]
  Call Extruder(399.40195)
  MoveL 10068 to (-39.95, 153.71, 144.49) mm, rotated rx 180 ry 0 rz 180 deg; joints [-53.036, -19.469, 100.708, 83.461, 53.537, -79.083]
  MoveL 10069 to (-39.95, 153.71, 144.49) mm, rotated rx 180 ry 0 rz 180 deg; joints [-53.036, -19.469, 100.708, 83.461, 53.537, -79.083]
  Call Extruder(399.53105)
  MoveL 10070 to (-40.02, 153.49, 144.49) mm, rotated rx 180 ry 0 rz 180 deg; joints [-53.022, -19.501, 100.73, 83.45, 53.525, -79.069]
  MoveL 10071 to (-40.02, 153.49, 144.49) mm, rotated rx 180 ry 0 rz 180 deg; joints [-53.022, -19.501, 100.73, 83.45, 53.525, -79.069]
  Call Extruder(399.64614)
  MoveL 10072 to (-40.06, 153.28, 144.49) mm, rotated rx 180 ry 0 rz 180 deg; joints [-53.007, -19.529, 100.749, 83.44, 53.511, -79.056]
  MoveL 10073 to (-40.06, 153.28, 144.49) mm, rotated rx 180 ry 0 rz 180 deg; joints [-53.007, -19.529, 100.749, 83.44, 53.511, -79.056]
  Call Extruder(399.76077)
  MoveL 10074 to (-40.11, 153.08, 144.49) mm, rotated rx -180 ry 0 rz 180 deg; joints [-52.993, -19.557, 100.768, 83.43, 53.498, -79.043]
  MoveL 10075 to (-40.11, 153.08, 144.49) mm, rotated rx -180 ry 0 rz 180 deg; joints [-52.993, -19.557, 100.768, 83.43, 53.498, -79.043]
  Call Extruder(399.87495)
  MoveL 10076 to (-40.15, 152.88, 144.49) mm, rotated rx 180 ry 0 rz 180 deg; joints [-52.978, -19.584, 100.787, 83.42, 53.485, -79.03]
  MoveL 10077 to (-40.15, 152.88, 144.49) mm, rotated rx 180 ry 0 rz 180 deg; joints [-52.978, -19.584, 100.787, 83.42, 53.485, -79.03]
  Call Extruder(399.98868)
  MoveL 10078 to (-40.2, 152.67, 144.49) mm, rotated rx -180 ry 0 rz 180 deg; joints [-52.963, -19.612, 100.806, 83.41, 53.471, -79.017]
  MoveL 10079 to (-40.2, 152.67, 144.49) mm, rotated rx -180 ry 0 rz 180 deg; joints [-52.963, -19.612, 100.806, 83.41, 53.471, -79.017]
  Call Extruder(400.11411)
  MoveL 10080 to (-40.24, 152.45, 144.49) mm, rotated rx 180 ry 0 rz 180 deg; joints [-52.946, -19.643, 100.827, 83.399, 53.456, -79.002]
  MoveL 10081 to (-40.24, 152.45, 144.49) mm, rotated rx 180 ry 0 rz 180 deg; joints [-52.946, -19.643, 100.827, 83.399, 53.456, -79.002]
  Call Extruder(400.25109)
  MoveL 10082 to (-40.29, 152.2, 144.49) mm, rotated rx 180 ry 0 rz 180 deg; joints [-52.928, -19.676, 100.85, 83.387, 53.439, -78.987]
  MoveL 10083 to (-40.29, 152.2, 144.49) mm, rotated rx 180 ry 0 rz 180 deg; joints [-52.928, -19.676, 100.85, 83.387, 53.439, -78.987]
  Call Extruder(400.38745)
  MoveL 10084 to (-40.34, 151.95, 144.49) mm, rotated rx 180 ry 0 rz 180 deg; joints [-52.909, -19.71, 100.872, 83.375, 53.421, -78.971]
  MoveL 10085 to (-40.34, 151.95, 144.49) mm, rotated rx 180 ry 0 rz 180 deg; joints [-52.909, -19.71, 100.872, 83.375, 53.421, -78.971]
  Call Extruder(400.52321)
  MoveL 10086 to (-40.39, 151.7, 144.49) mm, rotated rx 180 ry 0 rz 180 deg; joints [-52.89, -19.743, 100.895, 83.362, 53.404, -78.955]
  MoveL 10087 to (-40.39, 151.7, 144.49) mm, rotated rx 180 ry 0 rz 180 deg; joints [-52.89, -19.743, 100.895, 83.362, 53.404, -78.955]
  Call Extruder(400.65835)
  MoveL 10088 to (-40.44, 151.45, 144.49) mm, rotated rx 180 ry 0 rz 180 deg; joints [-52.871, -19.777, 100.918, 83.35, 53.387, -78.939]
  MoveL 10089 to (-40.44, 151.45, 144.49) mm, rotated rx 180 ry 0 rz 180 deg; joints [-52.871, -19.777, 100.918, 83.35, 53.387, -78.939]
  Call Extruder(400.79289)
  MoveL 10090 to (-40.49, 151.2, 144.49) mm, rotated rx 180 ry 0 rz 180 deg; joints [-52.853, -19.81, 100.941, 83.338, 53.37, -78.923]
  MoveL 10091 to (-40.49, 151.2, 144.49) mm, rotated rx 180 ry 0 rz 180 deg; joints [-52.853, -19.81, 100.941, 83.338, 53.37, -78.923]
  Call Extruder(400.92681)
  MoveL 10092 to (-40.54, 150.95, 144.49) mm, rotated rx -180 ry 0 rz 180 deg; joints [-52.834, -19.843, 100.963, 83.325, 53.352, -78.907]
  MoveL 10093 to (-40.54, 150.95, 144.49) mm, rotated rx -180 ry 0 rz 180 deg; joints [-52.834, -19.843, 100.963, 83.325, 53.352, -78.907]
  Call Extruder(401.07467)
  MoveL 10094 to (-40.59, 150.67, 144.49) mm, rotated rx -180 ry 0 rz 180 deg; joints [-52.812, -19.88, 100.988, 83.311, 53.332, -78.89]
  MoveL 10095 to (-40.59, 150.67, 144.49) mm, rotated rx -180 ry 0 rz 180 deg; joints [-52.812, -19.88, 100.988, 83.311, 53.332, -78.89]
  Call Extruder(401.23639)
  MoveL 10096 to (-40.64, 150.37, 144.49) mm, rotated rx 180 ry 0 rz 180 deg; joints [-52.787, -19.92, 101.015, 83.296, 53.31, -78.87]
  MoveL 10097 to (-40.64, 150.37, 144.49) mm, rotated rx 180 ry 0 rz 180 deg; joints [-52.787, -19.92, 101.015, 83.296, 53.31, -78.87]
  Call Extruder(401.39739)
  MoveL 10098 to (-40.69, 150.06, 144.49) mm, rotated rx 180 ry 0 rz 180 deg; joints [-52.762, -19.96, 101.042, 83.28, 53.287, -78.851]
  MoveL 10099 to (-40.69, 150.06, 144.49) mm, rotated rx 180 ry 0 rz 180 deg; joints [-52.762, -19.96, 101.042, 83.28, 53.287, -78.851]
  Call Extruder(401.55766)
  MoveL 10100 to (-40.74, 149.76, 144.49) mm, rotated rx 180 ry 0 rz 180 deg; joints [-52.737, -20, 101.069, 83.265, 53.264, -78.831]
  MoveL 10101 to (-40.74, 149.76, 144.49) mm, rotated rx 180 ry 0 rz 180 deg; joints [-52.737, -20, 101.069, 83.265, 53.264, -78.831]
  Call Extruder(401.71721)
  MoveL 10102 to (-40.78, 149.45, 144.49) mm, rotated rx 180 ry 0 rz 180 deg; joints [-52.712, -20.039, 101.096, 83.249, 53.241, -78.811]
  MoveL 10103 to (-40.78, 149.45, 144.49) mm, rotated rx 180 ry 0 rz 180 deg; joints [-52.712, -20.039, 101.096, 83.249, 53.241, -78.811]
  Call Extruder(401.87602)
  MoveL 10104 to (-40.83, 149.14, 144.49) mm, rotated rx -180 ry 0 rz 180 deg; joints [-52.687, -20.079, 101.123, 83.233, 53.218, -78.792]
  MoveL 10105 to (-40.83, 149.14, 144.49) mm, rotated rx -180 ry 0 rz 180 deg; joints [-52.687, -20.079, 101.123, 83.233, 53.218, -78.792]
  Call Extruder(402.05468)
  MoveL 10106 to (-40.88, 148.8, 144.49) mm, rotated rx -180 ry 0 rz 180 deg; joints [-52.658, -20.124, 101.153, 83.216, 53.191, -78.77]
  MoveL 10107 to (-40.88, 148.8, 144.49) mm, rotated rx -180 ry 0 rz 180 deg; joints [-52.658, -20.124, 101.153, 83.216, 53.191, -78.77]
  Call Extruder(402.25313)
  MoveL 10108 to (-40.92, 148.41, 144.49) mm, rotated rx -180 ry 0 rz 180 deg; joints [-52.624, -20.173, 101.186, 83.195, 53.159, -78.745]
  MoveL 10109 to (-40.92, 148.41, 144.49) mm, rotated rx -180 ry 0 rz 180 deg; joints [-52.624, -20.173, 101.186, 83.195, 53.159, -78.745]
  Call Extruder(402.45070)
  MoveL 10110 to (-40.97, 148.02, 144.49) mm, rotated rx 180 ry 0 rz -180 deg; joints [-52.59, -20.222, 101.219, 83.175, 53.128, -78.72]
  MoveL 10111 to (-40.97, 148.02, 144.49) mm, rotated rx 180 ry 0 rz -180 deg; joints [-52.59, -20.222, 101.219, 83.175, 53.128, -78.72]
  Call Extruder(402.64741)
  MoveL 10112 to (-41.02, 147.64, 144.49) mm, rotated rx 180 ry 0 rz 180 deg; joints [-52.556, -20.271, 101.252, 83.155, 53.096, -78.695]
  MoveL 10113 to (-41.02, 147.64, 144.49) mm, rotated rx 180 ry 0 rz 180 deg; joints [-52.556, -20.271, 101.252, 83.155, 53.096, -78.695]
  Call Extruder(402.84324)
  MoveL 10114 to (-41.06, 147.25, 144.49) mm, rotated rx -180 ry 0 rz 180 deg; joints [-52.521, -20.32, 101.285, 83.135, 53.064, -78.67]
  MoveL 10115 to (-41.06, 147.25, 144.49) mm, rotated rx -180 ry 0 rz 180 deg; joints [-52.521, -20.32, 101.285, 83.135, 53.064, -78.67]
  Call Extruder(403.13864)
  MoveL 10116 to (-41.11, 146.66, 144.49) mm, rotated rx 180 ry 0 rz 180 deg; joints [-52.466, -20.392, 101.334, 83.103, 53.013, -78.632]
  MoveL 10117 to (-41.11, 146.66, 144.49) mm, rotated rx 180 ry 0 rz 180 deg; joints [-52.466, -20.392, 101.334, 83.103, 53.013, -78.632]
  Call Extruder(403.43270)
  MoveL 10118 to (-41.16, 146.07, 144.49) mm, rotated rx 180 ry 0 rz 180 deg; joints [-52.411, -20.464, 101.382, 83.072, 52.962, -78.594]
  MoveL 10119 to (-41.16, 146.07, 144.49) mm, rotated rx 180 ry 0 rz 180 deg; joints [-52.411, -20.464, 101.382, 83.072, 52.962, -78.594]
  Call Extruder(403.72544)
  MoveL 10120 to (-41.2, 145.48, 144.49) mm, rotated rx 180 ry 0 rz 180 deg; joints [-52.355, -20.537, 101.431, 83.04, 52.91, -78.556]
  MoveL 10121 to (-41.2, 145.48, 144.49) mm, rotated rx 180 ry 0 rz 180 deg; joints [-52.355, -20.537, 101.431, 83.04, 52.91, -78.556]
  Call Extruder(404.29889)
  MoveL 10122 to (-41.25, 144.32, 144.49) mm, rotated rx 180 ry 0 rz 180 deg; joints [-52.239, -20.675, 101.523, 82.976, 52.802, -78.481]
  MoveL 10123 to (-41.25, 144.32, 144.49) mm, rotated rx 180 ry 0 rz 180 deg; joints [-52.239, -20.675, 101.523, 82.976, 52.802, -78.481]
  Call Extruder(405.01285)
  MoveL 10124 to (-41.29, 142.86, 144.49) mm, rotated rx 180 ry 0 rz 180 deg; joints [-52.09, -20.846, 101.636, 82.895, 52.663, -78.387]
  Call Extruder(447.07768)
  MoveL 10125 to (-41.29, 57.14, 144.49) mm, rotated rx 180 ry 0 rz 180 deg; joints [-40.759, -29.838, 106.937, 75.477, 42.409, -70.667]
  Call Extruder(447.50624)
  MoveL 10126 to (-41.27, 56.26, 144.49) mm, rotated rx 180 ry 0 rz -180 deg; joints [-40.614, -29.917, 106.977, 75.365, 42.283, -70.559]
  MoveL 10127 to (-41.27, 56.26, 144.49) mm, rotated rx 180 ry 0 rz -180 deg; joints [-40.614, -29.917, 106.977, 75.365, 42.283, -70.559]
  Call Extruder(448.07969)
  MoveL 10128 to (-41.23, 55.1, 144.49) mm, rotated rx 180 ry 0 rz 180 deg; joints [-40.419, -30.02, 107.03, 75.215, 42.111, -70.416]
  MoveL 10129 to (-41.23, 55.1, 144.49) mm, rotated rx 180 ry 0 rz 180 deg; joints [-40.419, -30.02, 107.03, 75.215, 42.111, -70.416]
  Call Extruder(448.51400)
  MoveL 10130 to (-41.18, 54.23, 144.49) mm, rotated rx 180 ry 0 rz 180 deg; joints [-40.269, -30.095, 107.069, 75.1, 41.979, -70.306]
  MoveL 10131 to (-41.18, 54.23, 144.49) mm, rotated rx 180 ry 0 rz 180 deg; joints [-40.269, -30.095, 107.069, 75.1, 41.979, -70.306]
  Call Extruder(448.80807)
  MoveL 10132 to (-41.13, 53.64, 144.49) mm, rotated rx 180 ry 0 rz 180 deg; joints [-40.165, -30.144, 107.094, 75.022, 41.888, -70.233]
  MoveL 10133 to (-41.13, 53.64, 144.49) mm, rotated rx 180 ry 0 rz 180 deg; joints [-40.165, -30.144, 107.094, 75.022, 41.888, -70.233]
  Call Extruder(449.10346)
  MoveL 10134 to (-41.09, 53.05, 144.49) mm, rotated rx 180 ry 0 rz 180 deg; joints [-40.062, -30.193, 107.119, 74.944, 41.797, -70.159]
  MoveL 10135 to (-41.09, 53.05, 144.49) mm, rotated rx 180 ry 0 rz 180 deg; joints [-40.062, -30.193, 107.119, 74.944, 41.797, -70.159]
  Call Extruder(449.34970)
  MoveL 10136 to (-41.04, 52.56, 144.49) mm, rotated rx 180 ry 0 rz 180 deg; joints [-39.975, -30.233, 107.139, 74.878, 41.72, -70.098]
  MoveL 10137 to (-41.04, 52.56, 144.49) mm, rotated rx 180 ry 0 rz 180 deg; joints [-39.975, -30.233, 107.139, 74.878, 41.72, -70.098]
  Call Extruder(449.54640)
  MoveL 10138 to (-40.99, 52.17, 144.49) mm, rotated rx -180 ry 0 rz 180 deg; joints [-39.904, -30.263, 107.154, 74.826, 41.658, -70.049]
  MoveL 10139 to (-40.99, 52.17, 144.49) mm, rotated rx -180 ry 0 rz 180 deg; joints [-39.904, -30.263, 107.154, 74.826, 41.658, -70.049]
  Call Extruder(449.74398)
  MoveL 10140 to (-40.95, 51.78, 144.49) mm, rotated rx 180 ry 0 rz 180 deg; joints [-39.833, -30.293, 107.17, 74.773, 41.595, -70]
  MoveL 10141 to (-40.95, 51.78, 144.49) mm, rotated rx 180 ry 0 rz 180 deg; joints [-39.833, -30.293, 107.17, 74.773, 41.595, -70]
  Call Extruder(449.94242)
  MoveL 10142 to (-40.9, 51.4, 144.49) mm, rotated rx 180 ry 0 rz 180 deg; joints [-39.763, -30.323, 107.185, 74.721, 41.533, -69.951]
  MoveL 10143 to (-40.9, 51.4, 144.49) mm, rotated rx 180 ry 0 rz 180 deg; joints [-39.763, -30.323, 107.185, 74.721, 41.533, -69.951]
  Call Extruder(450.14173)
  MoveL 10144 to (-40.86, 51.01, 144.49) mm, rotated rx 180 ry 0 rz 180 deg; joints [-39.692, -30.354, 107.2, 74.668, 41.47, -69.902]
  MoveL 10145 to (-40.86, 51.01, 144.49) mm, rotated rx 180 ry 0 rz 180 deg; joints [-39.692, -30.354, 107.2, 74.668, 41.47, -69.902]
  Call Extruder(450.30055)
  MoveL 10146 to (-40.81, 50.7, 144.49) mm, rotated rx -180 ry 0 rz 180 deg; joints [-39.634, -30.376, 107.212, 74.626, 41.419, -69.863]
  MoveL 10147 to (-40.81, 50.7, 144.49) mm, rotated rx -180 ry 0 rz 180 deg; joints [-39.634, -30.376, 107.212, 74.626, 41.419, -69.863]
  Call Extruder(450.46009)
  MoveL 10148 to (-40.76, 50.4, 144.49) mm, rotated rx 180 ry 0 rz -180 deg; joints [-39.576, -30.398, 107.223, 74.583, 41.367, -69.825]
  MoveL 10149 to (-40.76, 50.4, 144.49) mm, rotated rx 180 ry 0 rz -180 deg; joints [-39.576, -30.398, 107.223, 74.583, 41.367, -69.825]
  Call Extruder(450.62036)
